TEXTLIST S2_Alarms
  0 = 'S2 0 Row 1 Failed To Advance.. Check Qxxx.x Default' | German: 'S2 0 Row 1 Failed To Advance.. Check Qxxx.x German' | French: 'S2 0 Row 1 Failed To Advance.. Check Qxxx.x French'
  1 = 'S2 1 Row 1 Failed To Return.. Check Qxxx.x Default' | German: 'S2 1 Row 1 Failed To Return.. Check Qxxx.x German' | French: 'S2 1 Row 1 Failed To Return.. Check Qxxx.x French'
  2 = 'S2 2 Row 1 Lost Advance Position... Check Ixxx.x Default' | German: 'S2 2 Row 1 Lost Advance Position... Check Ixxx.x German' | French: 'S2 2 Row 1 Lost Advance Position... Check Ixxx.x French'
  3 = 'S2 3 Row 1 Lost Return Position... Check Ixxx.x Default' | German: 'S2 3 Row 1 Lost Return Position... Check Ixxx.x German' | French: 'S2 3 Row 1 Lost Return Position... Check Ixxx.x French'
  4 = 'S2 4 Row 1 Switch Fault... Check Ixxx.x / Ixxx.x Default' | German: 'S2 4 Row 1 Switch Fault... Check Ixxx.x / Ixxx.x German' | French: 'S2 4 Row 1 Switch Fault... Check Ixxx.x / Ixxx.x French'
  5 = 'S2 5 Row 1 Spare Message Default' | German: 'S2 5 Row 1 Spare Message German' | French: 'S2 5 Row 1 Spare Message French'
  6 = 'S2 6 Row 1 Spare Message Default' | German: 'S2 6 Row 1 Spare Message German' | French: 'S2 6 Row 1 Spare Message French'
  7 = 'S2 7 Row 1 Spare Message Default' | German: 'S2 7 Row 1 Spare Message German' | French: 'S2 7 Row 1 Spare Message French'
  8 = 'S2 8 Row 1 Spare Message Default' | German: 'S2 8 Row 1 Spare Message German' | French: 'S2 8 Row 1 Spare Message French'
  9 = 'S2 9 Row 1 Spare Message Default' | German: 'S2 9 Row 1 Spare Message German' | French: 'S2 9 Row 1 Spare Message French'
  10 = 'S2 10 Row 2 Failed To Advance.. Check Qxxx.x Default' | German: 'S2 10 Row 2 Failed To Advance.. Check Qxxx.x German' | French: 'S2 10 Row 2 Failed To Advance.. Check Qxxx.x French'
  11 = 'S2 11 Row 2 Failed To Return.. Check Qxxx.x Default' | German: 'S2 11 Row 2 Failed To Return.. Check Qxxx.x German' | French: 'S2 11 Row 2 Failed To Return.. Check Qxxx.x French'
  12 = 'S2 12 Row 2 Lost Advance Position... Check Ixxx.x Default' | German: 'S2 12 Row 2 Lost Advance Position... Check Ixxx.x German' | French: 'S2 12 Row 2 Lost Advance Position... Check Ixxx.x French'
  13 = 'S2 13 Row 2 Lost Return Position... Check Ixxx.x Default' | German: 'S2 13 Row 2 Lost Return Position... Check Ixxx.x German' | French: 'S2 13 Row 2 Lost Return Position... Check Ixxx.x French'
  14 = 'S2 14 Row 2 Switch Fault... Check Ixxx.x / Ixxx.x Default' | German: 'S2 14 Row 2 Switch Fault... Check Ixxx.x / Ixxx.x German' | French: 'S2 14 Row 2 Switch Fault... Check Ixxx.x / Ixxx.x French'
  15 = 'S2 15 Row 2 Spare Message Default' | German: 'S2 15 Row 2 Spare Message German' | French: 'S2 15 Row 2 Spare Message French'
  16 = 'S2 16 Row 2 Spare Message Default' | German: 'S2 16 Row 2 Spare Message German' | French: 'S2 16 Row 2 Spare Message French'
  17 = 'S2 17 Row 2 Spare Message Default' | German: 'S2 17 Row 2 Spare Message German' | French: 'S2 17 Row 2 Spare Message French'
  18 = 'S2 18 Row 2 Spare Message Default' | German: 'S2 18 Row 2 Spare Message German' | French: 'S2 18 Row 2 Spare Message French'
  19 = 'S2 19 Row 2 Spare Message Default' | German: 'S2 19 Row 2 Spare Message German' | French: 'S2 19 Row 2 Spare Message French'
  20 = 'S2 20 Row 3 Failed To Advance.. Check Qxxx.x Default' | German: 'S2 20 Row 3 Failed To Advance.. Check Qxxx.x German' | French: 'S2 20 Row 3 Failed To Advance.. Check Qxxx.x French'
  21 = 'S2 21 Row 3 Failed To Return.. Check Qxxx.x Default' | German: 'S2 21 Row 3 Failed To Return.. Check Qxxx.x German' | French: 'S2 21 Row 3 Failed To Return.. Check Qxxx.x French'
  22 = 'S2 22 Row 3 Lost Advance Position... Check Ixxx.x Default' | German: 'S2 22 Row 3 Lost Advance Position... Check Ixxx.x German' | French: 'S2 22 Row 3 Lost Advance Position... Check Ixxx.x French'
  23 = 'S2 23 Row 3 Lost Return Position... Check Ixxx.x Default' | German: 'S2 23 Row 3 Lost Return Position... Check Ixxx.x German' | French: 'S2 23 Row 3 Lost Return Position... Check Ixxx.x French'
  24 = 'S2 24 Row 3 Switch Fault... Check Ixxx.x / Ixxx.x Default' | German: 'S2 24 Row 3 Switch Fault... Check Ixxx.x / Ixxx.x German' | French: 'S2 24 Row 3 Switch Fault... Check Ixxx.x / Ixxx.x French'
  25 = 'S2 25 Row 3 Spare Message Default' | German: 'S2 25 Row 3 Spare Message German' | French: 'S2 25 Row 3 Spare Message French'
  26 = 'S2 26 Row 3 Spare Message Default' | German: 'S2 26 Row 3 Spare Message German' | French: 'S2 26 Row 3 Spare Message French'
  27 = 'S2 27 Row 3 Spare Message Default' | German: 'S2 27 Row 3 Spare Message German' | French: 'S2 27 Row 3 Spare Message French'
  28 = 'S2 28 Row 3 Spare Message Default' | German: 'S2 28 Row 3 Spare Message German' | French: 'S2 28 Row 3 Spare Message French'
  29 = 'S2 29 Row 3 Spare Message Default' | German: 'S2 29 Row 3 Spare Message German' | French: 'S2 29 Row 3 Spare Message French'
  30 = 'S2 30 Row 4 Failed To Advance.. Check Qxxx.x Default' | German: 'S2 30 Row 4 Failed To Advance.. Check Qxxx.x German' | French: 'S2 30 Row 4 Failed To Advance.. Check Qxxx.x French'
  31 = 'S2 31 Row 4 Failed To Return.. Check Qxxx.x Default' | German: 'S2 31 Row 4 Failed To Return.. Check Qxxx.x German' | French: 'S2 31 Row 4 Failed To Return.. Check Qxxx.x French'
  32 = 'S2 32 Row 4 Lost Advance Position... Check Ixxx.x Default' | German: 'S2 32 Row 4 Lost Advance Position... Check Ixxx.x German' | French: 'S2 32 Row 4 Lost Advance Position... Check Ixxx.x French'
  33 = 'S2 33 Row 4 Lost Return Position... Check Ixxx.x Default' | German: 'S2 33 Row 4 Lost Return Position... Check Ixxx.x German' | French: 'S2 33 Row 4 Lost Return Position... Check Ixxx.x French'
  34 = 'S2 34 Row 4 Switch Fault... Check Ixxx.x / Ixxx.x Default' | German: 'S2 34 Row 4 Switch Fault... Check Ixxx.x / Ixxx.x German' | French: 'S2 34 Row 4 Switch Fault... Check Ixxx.x / Ixxx.x French'
  35 = 'S2 35 Row 4 Spare Message Default' | German: 'S2 35 Row 4 Spare Message German' | French: 'S2 35 Row 4 Spare Message French'
  36 = 'S2 36 Row 4 Spare Message Default' | German: 'S2 36 Row 4 Spare Message German' | French: 'S2 36 Row 4 Spare Message French'
  37 = 'S2 37 Row 4 Spare Message Default' | German: 'S2 37 Row 4 Spare Message German' | French: 'S2 37 Row 4 Spare Message French'
  38 = 'S2 38 Row 4 Spare Message Default' | German: 'S2 38 Row 4 Spare Message German' | French: 'S2 38 Row 4 Spare Message French'
  39 = 'S2 39 Row 4 Spare Message Default' | German: 'S2 39 Row 4 Spare Message German' | French: 'S2 39 Row 4 Spare Message French'
  40 = 'S2 40 Row 5 Failed To Advance.. Check Qxxx.x Default' | German: 'S2 40 Row 5 Failed To Advance.. Check Qxxx.x German' | French: 'S2 40 Row 5 Failed To Advance.. Check Qxxx.x French'
  41 = 'S2 41 Row 5 Failed To Return.. Check Qxxx.x Default' | German: 'S2 41 Row 5 Failed To Return.. Check Qxxx.x German' | French: 'S2 41 Row 5 Failed To Return.. Check Qxxx.x French'
  42 = 'S2 42 Row 5 Lost Advance Position... Check Ixxx.x Default' | German: 'S2 42 Row 5 Lost Advance Position... Check Ixxx.x German' | French: 'S2 42 Row 5 Lost Advance Position... Check Ixxx.x French'
  43 = 'S2 43 Row 5 Lost Return Position... Check Ixxx.x Default' | German: 'S2 43 Row 5 Lost Return Position... Check Ixxx.x German' | French: 'S2 43 Row 5 Lost Return Position... Check Ixxx.x French'
  44 = 'S2 44 Row 5 Switch Fault... Check Ixxx.x / Ixxx.x Default' | German: 'S2 44 Row 5 Switch Fault... Check Ixxx.x / Ixxx.x German' | French: 'S2 44 Row 5 Switch Fault... Check Ixxx.x / Ixxx.x French'
  45 = 'S2 45 Row 5 Spare Message Default' | German: 'S2 45 Row 5 Spare Message German' | French: 'S2 45 Row 5 Spare Message French'
  46 = 'S2 46 Row 5 Spare Message Default' | German: 'S2 46 Row 5 Spare Message German' | French: 'S2 46 Row 5 Spare Message French'
  47 = 'S2 47 Row 5 Spare Message Default' | German: 'S2 47 Row 5 Spare Message German' | French: 'S2 47 Row 5 Spare Message French'
  48 = 'S2 48 Row 5 Spare Message Default' | German: 'S2 48 Row 5 Spare Message German' | French: 'S2 48 Row 5 Spare Message French'
  49 = 'S2 49 Row 5 Spare Message Default' | German: 'S2 49 Row 5 Spare Message German' | French: 'S2 49 Row 5 Spare Message French'
  50 = 'S2 50 Row 6 Failed To Advance.. Check Qxxx.x Default' | German: 'S2 50 Row 6 Failed To Advance.. Check Qxxx.x German' | French: 'S2 50 Row 6 Failed To Advance.. Check Qxxx.x French'
  51 = 'S2 51 Row 6 Failed To Return.. Check Qxxx.x Default' | German: 'S2 51 Row 6 Failed To Return.. Check Qxxx.x German' | French: 'S2 51 Row 6 Failed To Return.. Check Qxxx.x French'
  52 = 'S2 52 Row 6 Lost Advance Position... Check Ixxx.x Default' | German: 'S2 52 Row 6 Lost Advance Position... Check Ixxx.x German' | French: 'S2 52 Row 6 Lost Advance Position... Check Ixxx.x French'
  53 = 'S2 53 Row 6 Lost Return Position... Check Ixxx.x Default' | German: 'S2 53 Row 6 Lost Return Position... Check Ixxx.x German' | French: 'S2 53 Row 6 Lost Return Position... Check Ixxx.x French'
  54 = 'S2 54 Row 6 Switch Fault... Check Ixxx.x / Ixxx.x Default' | German: 'S2 54 Row 6 Switch Fault... Check Ixxx.x / Ixxx.x German' | French: 'S2 54 Row 6 Switch Fault... Check Ixxx.x / Ixxx.x French'
  55 = 'S2 55 Row 6 Spare Message Default' | German: 'S2 55 Row 6 Spare Message German' | French: 'S2 55 Row 6 Spare Message French'
  56 = 'S2 56 Row 6 Spare Message Default' | German: 'S2 56 Row 6 Spare Message German' | French: 'S2 56 Row 6 Spare Message French'
  57 = 'S2 57 Row 6 Spare Message Default' | German: 'S2 57 Row 6 Spare Message German' | French: 'S2 57 Row 6 Spare Message French'
  58 = 'S2 58 Row 6 Spare Message Default' | German: 'S2 58 Row 6 Spare Message German' | French: 'S2 58 Row 6 Spare Message French'
  59 = 'S2 59 Row 6 Spare Message Default' | German: 'S2 59 Row 6 Spare Message German' | French: 'S2 59 Row 6 Spare Message French'
  60 = 'S2 60 Row 7 Failed To Advance.. Check Qxxx.x Default' | German: 'S2 60 Row 7 Failed To Advance.. Check Qxxx.x German' | French: 'S2 60 Row 7 Failed To Advance.. Check Qxxx.x French'
  61 = 'S2 61 Row 7 Failed To Return.. Check Qxxx.x Default' | German: 'S2 61 Row 7 Failed To Return.. Check Qxxx.x German' | French: 'S2 61 Row 7 Failed To Return.. Check Qxxx.x French'
  62 = 'S2 62 Row 7 Lost Advance Position... Check Ixxx.x Default' | German: 'S2 62 Row 7 Lost Advance Position... Check Ixxx.x German' | French: 'S2 62 Row 7 Lost Advance Position... Check Ixxx.x French'
  63 = 'S2 63 Row 7 Lost Return Position... Check Ixxx.x Default' | German: 'S2 63 Row 7 Lost Return Position... Check Ixxx.x German' | French: 'S2 63 Row 7 Lost Return Position... Check Ixxx.x French'
  64 = 'S2 64 Row 7 Switch Fault... Check Ixxx.x / Ixxx.x Default' | German: 'S2 64 Row 7 Switch Fault... Check Ixxx.x / Ixxx.x German' | French: 'S2 64 Row 7 Switch Fault... Check Ixxx.x / Ixxx.x French'
  65 = 'S2 65 Row 7 Spare Message Default' | German: 'S2 65 Row 7 Spare Message German' | French: 'S2 65 Row 7 Spare Message French'
  66 = 'S2 66 Row 7 Spare Message Default' | German: 'S2 66 Row 7 Spare Message German' | French: 'S2 66 Row 7 Spare Message French'
  67 = 'S2 67 Row 7 Spare Message Default' | German: 'S2 67 Row 7 Spare Message German' | French: 'S2 67 Row 7 Spare Message French'
  68 = 'S2 68 Row 7 Spare Message Default' | German: 'S2 68 Row 7 Spare Message German' | French: 'S2 68 Row 7 Spare Message French'
  69 = 'S2 69 Row 7 Spare Message Default' | German: 'S2 69 Row 7 Spare Message German' | French: 'S2 69 Row 7 Spare Message French'
  70 = 'S2 70 Row 8 Failed To Advance.. Check Qxxx.x Default' | German: 'S2 70 Row 8 Failed To Advance.. Check Qxxx.x German' | French: 'S2 70 Row 8 Failed To Advance.. Check Qxxx.x French'
  71 = 'S2 71 Row 8 Failed To Return.. Check Qxxx.x Default' | German: 'S2 71 Row 8 Failed To Return.. Check Qxxx.x German' | French: 'S2 71 Row 8 Failed To Return.. Check Qxxx.x French'
  72 = 'S2 72 Row 8 Lost Advance Position... Check Ixxx.x Default' | German: 'S2 72 Row 8 Lost Advance Position... Check Ixxx.x German' | French: 'S2 72 Row 8 Lost Advance Position... Check Ixxx.x French'
  73 = 'S2 73 Row 8 Lost Return Position... Check Ixxx.x Default' | German: 'S2 73 Row 8 Lost Return Position... Check Ixxx.x German' | French: 'S2 73 Row 8 Lost Return Position... Check Ixxx.x French'
  74 = 'S2 74 Row 8 Switch Fault... Check Ixxx.x / Ixxx.x Default' | German: 'S2 74 Row 8 Switch Fault... Check Ixxx.x / Ixxx.x German' | French: 'S2 74 Row 8 Switch Fault... Check Ixxx.x / Ixxx.x French'
  75 = 'S2 75 Row 8 Spare Message Default' | German: 'S2 75 Row 8 Spare Message German' | French: 'S2 75 Row 8 Spare Message French'
  76 = 'S2 76 Row 8 Spare Message Default' | German: 'S2 76 Row 8 Spare Message German' | French: 'S2 76 Row 8 Spare Message French'
  77 = 'S2 77 Row 8 Spare Message Default' | German: 'S2 77 Row 8 Spare Message German' | French: 'S2 77 Row 8 Spare Message French'
  78 = 'S2 78 Row 8 Spare Message Default' | German: 'S2 78 Row 8 Spare Message German' | French: 'S2 78 Row 8 Spare Message French'
  79 = 'S2 79 Row 8 Spare Message Default' | German: 'S2 79 Row 8 Spare Message German' | French: 'S2 79 Row 8 Spare Message French'
  80 = 'S2 80 Row 9 Failed To Advance.. Check Qxxx.x Default' | German: 'S2 80 Row 9 Failed To Advance.. Check Qxxx.x German' | French: 'S2 80 Row 9 Failed To Advance.. Check Qxxx.x French'
  81 = 'S2 81 Row 9 Failed To Return.. Check Qxxx.x Default' | German: 'S2 81 Row 9 Failed To Return.. Check Qxxx.x German' | French: 'S2 81 Row 9 Failed To Return.. Check Qxxx.x French'
  82 = 'S2 82 Row 9 Lost Advance Position... Check Ixxx.x Default' | German: 'S2 82 Row 9 Lost Advance Position... Check Ixxx.x German' | French: 'S2 82 Row 9 Lost Advance Position... Check Ixxx.x French'
  83 = 'S2 83 Row 9 Lost Return Position... Check Ixxx.x Default' | German: 'S2 83 Row 9 Lost Return Position... Check Ixxx.x German' | French: 'S2 83 Row 9 Lost Return Position... Check Ixxx.x French'
  84 = 'S2 84 Row 9 Switch Fault... Check Ixxx.x / Ixxx.x Default' | German: 'S2 84 Row 9 Switch Fault... Check Ixxx.x / Ixxx.x German' | French: 'S2 84 Row 9 Switch Fault... Check Ixxx.x / Ixxx.x French'
  85 = 'S2 85 Row 9 Spare Message Default' | German: 'S2 85 Row 9 Spare Message German' | French: 'S2 85 Row 9 Spare Message French'
  86 = 'S2 86 Row 9 Spare Message Default' | German: 'S2 86 Row 9 Spare Message German' | French: 'S2 86 Row 9 Spare Message French'
  87 = 'S2 87 Row 9 Spare Message Default' | German: 'S2 87 Row 9 Spare Message German' | French: 'S2 87 Row 9 Spare Message French'
  88 = 'S2 88 Row 9 Spare Message Default' | German: 'S2 88 Row 9 Spare Message German' | French: 'S2 88 Row 9 Spare Message French'
  89 = 'S2 89 Row 9 Spare Message Default' | German: 'S2 89 Row 9 Spare Message German' | French: 'S2 89 Row 9 Spare Message French'
  90 = 'S2 90 Row 10 Failed To Advance.. Check Qxxx.x Default' | German: 'S2 90 Row 10 Failed To Advance.. Check Qxxx.x German' | French: 'S2 90 Row 10 Failed To Advance.. Check Qxxx.x French'
  91 = 'S2 91 Row 10 Failed To Return.. Check Qxxx.x Default' | German: 'S2 91 Row 10 Failed To Return.. Check Qxxx.x German' | French: 'S2 91 Row 10 Failed To Return.. Check Qxxx.x French'
  92 = 'S2 92 Row 10 Lost Advance Position... Check Ixxx.x Default' | German: 'S2 92 Row 10 Lost Advance Position... Check Ixxx.x German' | French: 'S2 92 Row 10 Lost Advance Position... Check Ixxx.x French'
  93 = 'S2 93 Row 10 Lost Return Position... Check Ixxx.x Default' | German: 'S2 93 Row 10 Lost Return Position... Check Ixxx.x German' | French: 'S2 93 Row 10 Lost Return Position... Check Ixxx.x French'
  94 = 'S2 94 Row 10 Switch Fault... Check Ixxx.x / Ixxx.x Default' | German: 'S2 94 Row 10 Switch Fault... Check Ixxx.x / Ixxx.x German' | French: 'S2 94 Row 10 Switch Fault... Check Ixxx.x / Ixxx.x French'
  95 = 'S2 95 Row 10 Spare Message Default' | German: 'S2 95 Row 10 Spare Message German' | French: 'S2 95 Row 10 Spare Message French'
  96 = 'S2 96 Row 10 Spare Message Default' | German: 'S2 96 Row 10 Spare Message German' | French: 'S2 96 Row 10 Spare Message French'
  97 = 'S2 97 Row 10 Spare Message Default' | German: 'S2 97 Row 10 Spare Message German' | French: 'S2 97 Row 10 Spare Message French'
  98 = 'S2 98 Row 10 Spare Message Default' | German: 'S2 98 Row 10 Spare Message German' | French: 'S2 98 Row 10 Spare Message French'
  99 = 'S2 99 Row 10 Spare Message Default' | German: 'S2 99 Row 10 Spare Message German' | French: 'S2 99 Row 10 Spare Message French'
  100 = 'S2 100 Row 11 Failed To Advance.. Check Qxxx.x Default' | German: 'S2 100 Row 11 Failed To Advance.. Check Qxxx.x German' | French: 'S2 100 Row 11 Failed To Advance.. Check Qxxx.x French'
  101 = 'S2 101 Row 11 Failed To Return.. Check Qxxx.x Default' | German: 'S2 101 Row 11 Failed To Return.. Check Qxxx.x German' | French: 'S2 101 Row 11 Failed To Return.. Check Qxxx.x French'
  102 = 'S2 102 Row 11 Lost Advance Position... Check Ixxx.x Default' | German: 'S2 102 Row 11 Lost Advance Position... Check Ixxx.x German' | French: 'S2 102 Row 11 Lost Advance Position... Check Ixxx.x French'
  103 = 'S2 103 Row 11 Lost Return Position... Check Ixxx.x Default' | German: 'S2 103 Row 11 Lost Return Position... Check Ixxx.x German' | French: 'S2 103 Row 11 Lost Return Position... Check Ixxx.x French'
  104 = 'S2 104 Row 11 Switch Fault... Check Ixxx.x / Ixxx.x Default' | German: 'S2 104 Row 11 Switch Fault... Check Ixxx.x / Ixxx.x German' | French: 'S2 104 Row 11 Switch Fault... Check Ixxx.x / Ixxx.x French'
  105 = 'S2 105 Row 11 Spare Message Default' | German: 'S2 105 Row 11 Spare Message German' | French: 'S2 105 Row 11 Spare Message French'
  106 = 'S2 106 Row 11 Spare Message Default' | German: 'S2 106 Row 11 Spare Message German' | French: 'S2 106 Row 11 Spare Message French'
  107 = 'S2 107 Row 11 Spare Message Default' | German: 'S2 107 Row 11 Spare Message German' | French: 'S2 107 Row 11 Spare Message French'
  108 = 'S2 108 Row 11 Spare Message Default' | German: 'S2 108 Row 11 Spare Message German' | French: 'S2 108 Row 11 Spare Message French'
  109 = 'S2 109 Row 11 Spare Message Default' | German: 'S2 109 Row 11 Spare Message German' | French: 'S2 109 Row 11 Spare Message French'
  110 = 'S2 110 Row 12 Failed To Advance.. Check Qxxx.x Default' | German: 'S2 110 Row 12 Failed To Advance.. Check Qxxx.x German' | French: 'S2 110 Row 12 Failed To Advance.. Check Qxxx.x French'
  111 = 'S2 111 Row 12 Failed To Return.. Check Qxxx.x Default' | German: 'S2 111 Row 12 Failed To Return.. Check Qxxx.x German' | French: 'S2 111 Row 12 Failed To Return.. Check Qxxx.x French'
  112 = 'S2 112 Row 12 Lost Advance Position... Check Ixxx.x Default' | German: 'S2 112 Row 12 Lost Advance Position... Check Ixxx.x German' | French: 'S2 112 Row 12 Lost Advance Position... Check Ixxx.x French'
  113 = 'S2 113 Row 12 Lost Return Position... Check Ixxx.x Default' | German: 'S2 113 Row 12 Lost Return Position... Check Ixxx.x German' | French: 'S2 113 Row 12 Lost Return Position... Check Ixxx.x French'
  114 = 'S2 114 Row 12 Switch Fault... Check Ixxx.x / Ixxx.x Default' | German: 'S2 114 Row 12 Switch Fault... Check Ixxx.x / Ixxx.x German' | French: 'S2 114 Row 12 Switch Fault... Check Ixxx.x / Ixxx.x French'
  115 = 'S2 115 Row 12 Spare Message Default' | German: 'S2 115 Row 12 Spare Message German' | French: 'S2 115 Row 12 Spare Message French'
  116 = 'S2 116 Row 12 Spare Message Default' | German: 'S2 116 Row 12 Spare Message German' | French: 'S2 116 Row 12 Spare Message French'
  117 = 'S2 117 Row 12 Spare Message Default' | German: 'S2 117 Row 12 Spare Message German' | French: 'S2 117 Row 12 Spare Message French'
  118 = 'S2 118 Row 12 Spare Message Default' | German: 'S2 118 Row 12 Spare Message German' | French: 'S2 118 Row 12 Spare Message French'
  119 = 'S2 119 Row 12 Spare Message Default' | German: 'S2 119 Row 12 Spare Message German' | French: 'S2 119 Row 12 Spare Message French'
  120 = 'S2 120 Row 13 Failed To Advance.. Check Qxxx.x Default' | German: 'S2 120 Row 13 Failed To Advance.. Check Qxxx.x German' | French: 'S2 120 Row 13 Failed To Advance.. Check Qxxx.x French'
  121 = 'S2 121 Row 13 Failed To Return.. Check Qxxx.x Default' | German: 'S2 121 Row 13 Failed To Return.. Check Qxxx.x German' | French: 'S2 121 Row 13 Failed To Return.. Check Qxxx.x French'
  122 = 'S2 122 Row 13 Lost Advance Position... Check Ixxx.x Default' | German: 'S2 122 Row 13 Lost Advance Position... Check Ixxx.x German' | French: 'S2 122 Row 13 Lost Advance Position... Check Ixxx.x French'
  123 = 'S2 123 Row 13 Lost Return Position... Check Ixxx.x Default' | German: 'S2 123 Row 13 Lost Return Position... Check Ixxx.x German' | French: 'S2 123 Row 13 Lost Return Position... Check Ixxx.x French'
  124 = 'S2 124 Row 13 Switch Fault... Check Ixxx.x / Ixxx.x Default' | German: 'S2 124 Row 13 Switch Fault... Check Ixxx.x / Ixxx.x German' | French: 'S2 124 Row 13 Switch Fault... Check Ixxx.x / Ixxx.x French'
  125 = 'S2 125 Row 13 Spare Message Default' | German: 'S2 125 Row 13 Spare Message German' | French: 'S2 125 Row 13 Spare Message French'
  126 = 'S2 126 Row 13 Spare Message Default' | German: 'S2 126 Row 13 Spare Message German' | French: 'S2 126 Row 13 Spare Message French'
  127 = 'S2 127 Row 13 Spare Message Default' | German: 'S2 127 Row 13 Spare Message German' | French: 'S2 127 Row 13 Spare Message French'
  128 = 'S2 128 Row 13 Spare Message Default' | German: 'S2 128 Row 13 Spare Message German' | French: 'S2 128 Row 13 Spare Message French'
  129 = 'S2 129 Row 13 Spare Message Default' | German: 'S2 129 Row 13 Spare Message German' | French: 'S2 129 Row 13 Spare Message French'
  130 = 'S2 130 Row 14 Failed To Advance.. Check Qxxx.x Default' | German: 'S2 130 Row 14 Failed To Advance.. Check Qxxx.x German' | French: 'S2 130 Row 14 Failed To Advance.. Check Qxxx.x French'
  131 = 'S2 131 Row 14 Failed To Return.. Check Qxxx.x Default' | German: 'S2 131 Row 14 Failed To Return.. Check Qxxx.x German' | French: 'S2 131 Row 14 Failed To Return.. Check Qxxx.x French'
  132 = 'S2 132 Row 14 Lost Advance Position... Check Ixxx.x Default' | German: 'S2 132 Row 14 Lost Advance Position... Check Ixxx.x German' | French: 'S2 132 Row 14 Lost Advance Position... Check Ixxx.x French'
  133 = 'S2 133 Row 14 Lost Return Position... Check Ixxx.x Default' | German: 'S2 133 Row 14 Lost Return Position... Check Ixxx.x German' | French: 'S2 133 Row 14 Lost Return Position... Check Ixxx.x French'
  134 = 'S2 134 Row 14 Switch Fault... Check Ixxx.x / Ixxx.x Default' | German: 'S2 134 Row 14 Switch Fault... Check Ixxx.x / Ixxx.x German' | French: 'S2 134 Row 14 Switch Fault... Check Ixxx.x / Ixxx.x French'
  135 = 'S2 135 Row 14 Spare Message Default' | German: 'S2 135 Row 14 Spare Message German' | French: 'S2 135 Row 14 Spare Message French'
  136 = 'S2 136 Row 14 Spare Message Default' | German: 'S2 136 Row 14 Spare Message German' | French: 'S2 136 Row 14 Spare Message French'
  137 = 'S2 137 Row 14 Spare Message Default' | German: 'S2 137 Row 14 Spare Message German' | French: 'S2 137 Row 14 Spare Message French'
  138 = 'S2 138 Row 14 Spare Message Default' | German: 'S2 138 Row 14 Spare Message German' | French: 'S2 138 Row 14 Spare Message French'
  139 = 'S2 139 Row 14 Spare Message Default' | German: 'S2 139 Row 14 Spare Message German' | French: 'S2 139 Row 14 Spare Message French'
  140 = 'S2 140 Row 15 Failed To Advance.. Check Qxxx.x Default' | German: 'S2 140 Row 15 Failed To Advance.. Check Qxxx.x German' | French: 'S2 140 Row 15 Failed To Advance.. Check Qxxx.x French'
  141 = 'S2 141 Row 15 Failed To Return.. Check Qxxx.x Default' | German: 'S2 141 Row 15 Failed To Return.. Check Qxxx.x German' | French: 'S2 141 Row 15 Failed To Return.. Check Qxxx.x French'
  142 = 'S2 142 Row 15 Lost Advance Position... Check Ixxx.x Default' | German: 'S2 142 Row 15 Lost Advance Position... Check Ixxx.x German' | French: 'S2 142 Row 15 Lost Advance Position... Check Ixxx.x French'
  143 = 'S2 143 Row 15 Lost Return Position... Check Ixxx.x Default' | German: 'S2 143 Row 15 Lost Return Position... Check Ixxx.x German' | French: 'S2 143 Row 15 Lost Return Position... Check Ixxx.x French'
  144 = 'S2 144 Row 15 Switch Fault... Check Ixxx.x / Ixxx.x Default' | German: 'S2 144 Row 15 Switch Fault... Check Ixxx.x / Ixxx.x German' | French: 'S2 144 Row 15 Switch Fault... Check Ixxx.x / Ixxx.x French'
  145 = 'S2 145 Row 15 Spare Message Default' | German: 'S2 145 Row 15 Spare Message German' | French: 'S2 145 Row 15 Spare Message French'
  146 = 'S2 146 Row 15 Spare Message Default' | German: 'S2 146 Row 15 Spare Message German' | French: 'S2 146 Row 15 Spare Message French'
  147 = 'S2 147 Row 15 Spare Message Default' | German: 'S2 147 Row 15 Spare Message German' | French: 'S2 147 Row 15 Spare Message French'
  148 = 'S2 148 Row 15 Spare Message Default' | German: 'S2 148 Row 15 Spare Message German' | French: 'S2 148 Row 15 Spare Message French'
  149 = 'S2 149 Row 15 Spare Message Default' | German: 'S2 149 Row 15 Spare Message German' | French: 'S2 149 Row 15 Spare Message French'
  150 = 'S2 150 Row 16 Failed To Advance.. Check Qxxx.x Default' | German: 'S2 150 Row 16 Failed To Advance.. Check Qxxx.x German' | French: 'S2 150 Row 16 Failed To Advance.. Check Qxxx.x French'
  151 = 'S2 151 Row 16 Failed To Return.. Check Qxxx.x Default' | German: 'S2 151 Row 16 Failed To Return.. Check Qxxx.x German' | French: 'S2 151 Row 16 Failed To Return.. Check Qxxx.x French'
  152 = 'S2 152 Row 16 Lost Advance Position... Check Ixxx.x Default' | German: 'S2 152 Row 16 Lost Advance Position... Check Ixxx.x German' | French: 'S2 152 Row 16 Lost Advance Position... Check Ixxx.x French'
  153 = 'S2 153 Row 16 Lost Return Position... Check Ixxx.x Default' | German: 'S2 153 Row 16 Lost Return Position... Check Ixxx.x German' | French: 'S2 153 Row 16 Lost Return Position... Check Ixxx.x French'
  154 = 'S2 154 Row 16 Switch Fault... Check Ixxx.x / Ixxx.x Default' | German: 'S2 154 Row 16 Switch Fault... Check Ixxx.x / Ixxx.x German' | French: 'S2 154 Row 16 Switch Fault... Check Ixxx.x / Ixxx.x French'
  155 = 'S2 155 Row 16 Spare Message Default' | German: 'S2 155 Row 16 Spare Message German' | French: 'S2 155 Row 16 Spare Message French'
  156 = 'S2 156 Row 16 Spare Message Default' | German: 'S2 156 Row 16 Spare Message German' | French: 'S2 156 Row 16 Spare Message French'
  157 = 'S2 157 Row 16 Spare Message Default' | German: 'S2 157 Row 16 Spare Message German' | French: 'S2 157 Row 16 Spare Message French'
  158 = 'S2 158 Row 16 Spare Message Default' | German: 'S2 158 Row 16 Spare Message German' | French: 'S2 158 Row 16 Spare Message French'
  159 = 'S2 159 Row 16 Spare Message Default' | German: 'S2 159 Row 16 Spare Message German' | French: 'S2 159 Row 16 Spare Message French'
  160 = 'S2 160 Row 17 Failed To Advance.. Check Qxxx.x Default' | German: 'S2 160 Row 17 Failed To Advance.. Check Qxxx.x German' | French: 'S2 160 Row 17 Failed To Advance.. Check Qxxx.x French'
  161 = 'S2 161 Row 17 Failed To Return.. Check Qxxx.x Default' | German: 'S2 161 Row 17 Failed To Return.. Check Qxxx.x German' | French: 'S2 161 Row 17 Failed To Return.. Check Qxxx.x French'
  162 = 'S2 162 Row 17 Lost Advance Position... Check Ixxx.x Default' | German: 'S2 162 Row 17 Lost Advance Position... Check Ixxx.x German' | French: 'S2 162 Row 17 Lost Advance Position... Check Ixxx.x French'
  163 = 'S2 163 Row 17 Lost Return Position... Check Ixxx.x Default' | German: 'S2 163 Row 17 Lost Return Position... Check Ixxx.x German' | French: 'S2 163 Row 17 Lost Return Position... Check Ixxx.x French'
  164 = 'S2 164 Row 17 Switch Fault... Check Ixxx.x / Ixxx.x Default' | German: 'S2 164 Row 17 Switch Fault... Check Ixxx.x / Ixxx.x German' | French: 'S2 164 Row 17 Switch Fault... Check Ixxx.x / Ixxx.x French'
  165 = 'S2 165 Row 17 Spare Message Default' | German: 'S2 165 Row 17 Spare Message German' | French: 'S2 165 Row 17 Spare Message French'
  166 = 'S2 166 Row 17 Spare Message Default' | German: 'S2 166 Row 17 Spare Message German' | French: 'S2 166 Row 17 Spare Message French'
  167 = 'S2 167 Row 17 Spare Message Default' | German: 'S2 167 Row 17 Spare Message German' | French: 'S2 167 Row 17 Spare Message French'
  168 = 'S2 168 Row 17 Spare Message Default' | German: 'S2 168 Row 17 Spare Message German' | French: 'S2 168 Row 17 Spare Message French'
  169 = 'S2 169 Row 17 Spare Message Default' | German: 'S2 169 Row 17 Spare Message German' | French: 'S2 169 Row 17 Spare Message French'
  170 = 'S2 170 Row 18 Failed To Advance.. Check Qxxx.x Default' | German: 'S2 170 Row 18 Failed To Advance.. Check Qxxx.x German' | French: 'S2 170 Row 18 Failed To Advance.. Check Qxxx.x French'
  171 = 'S2 171 Row 18 Failed To Return.. Check Qxxx.x Default' | German: 'S2 171 Row 18 Failed To Return.. Check Qxxx.x German' | French: 'S2 171 Row 18 Failed To Return.. Check Qxxx.x French'
  172 = 'S2 172 Row 18 Lost Advance Position... Check Ixxx.x Default' | German: 'S2 172 Row 18 Lost Advance Position... Check Ixxx.x German' | French: 'S2 172 Row 18 Lost Advance Position... Check Ixxx.x French'
  173 = 'S2 173 Row 18 Lost Return Position... Check Ixxx.x Default' | German: 'S2 173 Row 18 Lost Return Position... Check Ixxx.x German' | French: 'S2 173 Row 18 Lost Return Position... Check Ixxx.x French'
  174 = 'S2 174 Row 18 Switch Fault... Check Ixxx.x / Ixxx.x Default' | German: 'S2 174 Row 18 Switch Fault... Check Ixxx.x / Ixxx.x German' | French: 'S2 174 Row 18 Switch Fault... Check Ixxx.x / Ixxx.x French'
  175 = 'S2 175 Row 18 Spare Message Default' | German: 'S2 175 Row 18 Spare Message German' | French: 'S2 175 Row 18 Spare Message French'
  176 = 'S2 176 Row 18 Spare Message Default' | German: 'S2 176 Row 18 Spare Message German' | French: 'S2 176 Row 18 Spare Message French'
  177 = 'S2 177 Row 18 Spare Message Default' | German: 'S2 177 Row 18 Spare Message German' | French: 'S2 177 Row 18 Spare Message French'
  178 = 'S2 178 Row 18 Spare Message Default' | German: 'S2 178 Row 18 Spare Message German' | French: 'S2 178 Row 18 Spare Message French'
  179 = 'S2 179 Row 18 Spare Message Default' | German: 'S2 179 Row 18 Spare Message German' | French: 'S2 179 Row 18 Spare Message French'
  180 = 'S2 180 Row 19 Failed To Advance.. Check Qxxx.x Default' | German: 'S2 180 Row 19 Failed To Advance.. Check Qxxx.x German' | French: 'S2 180 Row 19 Failed To Advance.. Check Qxxx.x French'
  181 = 'S2 181 Row 19 Failed To Return.. Check Qxxx.x Default' | German: 'S2 181 Row 19 Failed To Return.. Check Qxxx.x German' | French: 'S2 181 Row 19 Failed To Return.. Check Qxxx.x French'
  182 = 'S2 182 Row 19 Lost Advance Position... Check Ixxx.x Default' | German: 'S2 182 Row 19 Lost Advance Position... Check Ixxx.x German' | French: 'S2 182 Row 19 Lost Advance Position... Check Ixxx.x French'
  183 = 'S2 183 Row 19 Lost Return Position... Check Ixxx.x Default' | German: 'S2 183 Row 19 Lost Return Position... Check Ixxx.x German' | French: 'S2 183 Row 19 Lost Return Position... Check Ixxx.x French'
  184 = 'S2 184 Row 19 Switch Fault... Check Ixxx.x / Ixxx.x Default' | German: 'S2 184 Row 19 Switch Fault... Check Ixxx.x / Ixxx.x German' | French: 'S2 184 Row 19 Switch Fault... Check Ixxx.x / Ixxx.x French'
  185 = 'S2 185 Row 19 Spare Message Default' | German: 'S2 185 Row 19 Spare Message German' | French: 'S2 185 Row 19 Spare Message French'
  186 = 'S2 186 Row 19 Spare Message Default' | German: 'S2 186 Row 19 Spare Message German' | French: 'S2 186 Row 19 Spare Message French'
  187 = 'S2 187 Row 19 Spare Message Default' | German: 'S2 187 Row 19 Spare Message German' | French: 'S2 187 Row 19 Spare Message French'
  188 = 'S2 188 Row 19 Spare Message Default' | German: 'S2 188 Row 19 Spare Message German' | French: 'S2 188 Row 19 Spare Message French'
  189 = 'S2 189 Row 19 Spare Message Default' | German: 'S2 189 Row 19 Spare Message German' | French: 'S2 189 Row 19 Spare Message French'
  190 = 'S2 190 Row 20 Failed To Advance.. Check Qxxx.x Default' | German: 'S2 190 Row 20 Failed To Advance.. Check Qxxx.x German' | French: 'S2 190 Row 20 Failed To Advance.. Check Qxxx.x French'
  191 = 'S2 191 Row 20 Failed To Return.. Check Qxxx.x Default' | German: 'S2 191 Row 20 Failed To Return.. Check Qxxx.x German' | French: 'S2 191 Row 20 Failed To Return.. Check Qxxx.x French'
  192 = 'S2 192 Row 20 Lost Advance Position... Check Ixxx.x Default' | German: 'S2 192 Row 20 Lost Advance Position... Check Ixxx.x German' | French: 'S2 192 Row 20 Lost Advance Position... Check Ixxx.x French'
  193 = 'S2 193 Row 20 Lost Return Position... Check Ixxx.x Default' | German: 'S2 193 Row 20 Lost Return Position... Check Ixxx.x German' | French: 'S2 193 Row 20 Lost Return Position... Check Ixxx.x French'
  194 = 'S2 194 Row 20 Switch Fault... Check Ixxx.x / Ixxx.x Default' | German: 'S2 194 Row 20 Switch Fault... Check Ixxx.x / Ixxx.x German' | French: 'S2 194 Row 20 Switch Fault... Check Ixxx.x / Ixxx.x French'
  195 = 'S2 195 Row 20 Spare Message Default' | German: 'S2 195 Row 20 Spare Message German' | French: 'S2 195 Row 20 Spare Message French'
  196 = 'S2 196 Row 20 Spare Message Default' | German: 'S2 196 Row 20 Spare Message German' | French: 'S2 196 Row 20 Spare Message French'
  197 = 'S2 197 Row 20 Spare Message Default' | German: 'S2 197 Row 20 Spare Message German' | French: 'S2 197 Row 20 Spare Message French'
  198 = 'S2 198 Row 20 Spare Message Default' | German: 'S2 198 Row 20 Spare Message German' | French: 'S2 198 Row 20 Spare Message French'
  199 = 'S2 199 Row 20 Spare Message Default' | German: 'S2 199 Row 20 Spare Message German' | French: 'S2 199 Row 20 Spare Message French'
  200 = 'S2 200 Row 21 Failed To Advance.. Check Qxxx.x Default' | German: 'S2 200 Row 21 Failed To Advance.. Check Qxxx.x German' | French: 'S2 200 Row 21 Failed To Advance.. Check Qxxx.x French'
  201 = 'S2 201 Row 21 Failed To Return.. Check Qxxx.x Default' | German: 'S2 201 Row 21 Failed To Return.. Check Qxxx.x German' | French: 'S2 201 Row 21 Failed To Return.. Check Qxxx.x French'
  202 = 'S2 202 Row 21 Lost Advance Position... Check Ixxx.x Default' | German: 'S2 202 Row 21 Lost Advance Position... Check Ixxx.x German' | French: 'S2 202 Row 21 Lost Advance Position... Check Ixxx.x French'
  203 = 'S2 203 Row 21 Lost Return Position... Check Ixxx.x Default' | German: 'S2 203 Row 21 Lost Return Position... Check Ixxx.x German' | French: 'S2 203 Row 21 Lost Return Position... Check Ixxx.x French'
  204 = 'S2 204 Row 21 Switch Fault... Check Ixxx.x / Ixxx.x Default' | German: 'S2 204 Row 21 Switch Fault... Check Ixxx.x / Ixxx.x German' | French: 'S2 204 Row 21 Switch Fault... Check Ixxx.x / Ixxx.x French'
  205 = 'S2 205 Row 21 Spare Message Default' | German: 'S2 205 Row 21 Spare Message German' | French: 'S2 205 Row 21 Spare Message French'
  206 = 'S2 206 Row 21 Spare Message Default' | German: 'S2 206 Row 21 Spare Message German' | French: 'S2 206 Row 21 Spare Message French'
  207 = 'S2 207 Row 21 Spare Message Default' | German: 'S2 207 Row 21 Spare Message German' | French: 'S2 207 Row 21 Spare Message French'
  208 = 'S2 208 Row 21 Spare Message Default' | German: 'S2 208 Row 21 Spare Message German' | French: 'S2 208 Row 21 Spare Message French'
  209 = 'S2 209 Row 21 Spare Message Default' | German: 'S2 209 Row 21 Spare Message German' | French: 'S2 209 Row 21 Spare Message French'
  210 = 'S2 210 Row 22 Failed To Advance.. Check Qxxx.x Default' | German: 'S2 210 Row 22 Failed To Advance.. Check Qxxx.x German' | French: 'S2 210 Row 22 Failed To Advance.. Check Qxxx.x French'
  211 = 'S2 211 Row 22 Failed To Return.. Check Qxxx.x Default' | German: 'S2 211 Row 22 Failed To Return.. Check Qxxx.x German' | French: 'S2 211 Row 22 Failed To Return.. Check Qxxx.x French'
  212 = 'S2 212 Row 22 Lost Advance Position... Check Ixxx.x Default' | German: 'S2 212 Row 22 Lost Advance Position... Check Ixxx.x German' | French: 'S2 212 Row 22 Lost Advance Position... Check Ixxx.x French'
  213 = 'S2 213 Row 22 Lost Return Position... Check Ixxx.x Default' | German: 'S2 213 Row 22 Lost Return Position... Check Ixxx.x German' | French: 'S2 213 Row 22 Lost Return Position... Check Ixxx.x French'
  214 = 'S2 214 Row 22 Switch Fault... Check Ixxx.x / Ixxx.x Default' | German: 'S2 214 Row 22 Switch Fault... Check Ixxx.x / Ixxx.x German' | French: 'S2 214 Row 22 Switch Fault... Check Ixxx.x / Ixxx.x French'
  215 = 'S2 215 Row 22 Spare Message Default' | German: 'S2 215 Row 22 Spare Message German' | French: 'S2 215 Row 22 Spare Message French'
  216 = 'S2 216 Row 22 Spare Message Default' | German: 'S2 216 Row 22 Spare Message German' | French: 'S2 216 Row 22 Spare Message French'
  217 = 'S2 217 Row 22 Spare Message Default' | German: 'S2 217 Row 22 Spare Message German' | French: 'S2 217 Row 22 Spare Message French'
  218 = 'S2 218 Row 22 Spare Message Default' | German: 'S2 218 Row 22 Spare Message German' | French: 'S2 218 Row 22 Spare Message French'
  219 = 'S2 219 Row 22 Spare Message Default' | German: 'S2 219 Row 22 Spare Message German' | French: 'S2 219 Row 22 Spare Message French'
  220 = 'S2 220 Row 23 Failed To Advance.. Check Qxxx.x Default' | German: 'S2 220 Row 23 Failed To Advance.. Check Qxxx.x German' | French: 'S2 220 Row 23 Failed To Advance.. Check Qxxx.x French'
  221 = 'S2 221 Row 23 Failed To Return.. Check Qxxx.x Default' | German: 'S2 221 Row 23 Failed To Return.. Check Qxxx.x German' | French: 'S2 221 Row 23 Failed To Return.. Check Qxxx.x French'
  222 = 'S2 222 Row 23 Lost Advance Position... Check Ixxx.x Default' | German: 'S2 222 Row 23 Lost Advance Position... Check Ixxx.x German' | French: 'S2 222 Row 23 Lost Advance Position... Check Ixxx.x French'
  223 = 'S2 223 Row 23 Lost Return Position... Check Ixxx.x Default' | German: 'S2 223 Row 23 Lost Return Position... Check Ixxx.x German' | French: 'S2 223 Row 23 Lost Return Position... Check Ixxx.x French'
  224 = 'S2 224 Row 23 Switch Fault... Check Ixxx.x / Ixxx.x Default' | German: 'S2 224 Row 23 Switch Fault... Check Ixxx.x / Ixxx.x German' | French: 'S2 224 Row 23 Switch Fault... Check Ixxx.x / Ixxx.x French'
  225 = 'S2 225 Row 23 Spare Message Default' | German: 'S2 225 Row 23 Spare Message German' | French: 'S2 225 Row 23 Spare Message French'
  226 = 'S2 226 Row 23 Spare Message Default' | German: 'S2 226 Row 23 Spare Message German' | French: 'S2 226 Row 23 Spare Message French'
  227 = 'S2 227 Row 23 Spare Message Default' | German: 'S2 227 Row 23 Spare Message German' | French: 'S2 227 Row 23 Spare Message French'
  228 = 'S2 228 Row 23 Spare Message Default' | German: 'S2 228 Row 23 Spare Message German' | French: 'S2 228 Row 23 Spare Message French'
  229 = 'S2 229 Row 23 Spare Message Default' | German: 'S2 229 Row 23 Spare Message German' | French: 'S2 229 Row 23 Spare Message French'
  230 = 'S2 230 Row 24 Failed To Advance.. Check Qxxx.x Default' | German: 'S2 230 Row 24 Failed To Advance.. Check Qxxx.x German' | French: 'S2 230 Row 24 Failed To Advance.. Check Qxxx.x French'
  231 = 'S2 231 Row 24 Failed To Return.. Check Qxxx.x Default' | German: 'S2 231 Row 24 Failed To Return.. Check Qxxx.x German' | French: 'S2 231 Row 24 Failed To Return.. Check Qxxx.x French'
  232 = 'S2 232 Row 24 Lost Advance Position... Check Ixxx.x Default' | German: 'S2 232 Row 24 Lost Advance Position... Check Ixxx.x German' | French: 'S2 232 Row 24 Lost Advance Position... Check Ixxx.x French'
  233 = 'S2 233 Row 24 Lost Return Position... Check Ixxx.x Default' | German: 'S2 233 Row 24 Lost Return Position... Check Ixxx.x German' | French: 'S2 233 Row 24 Lost Return Position... Check Ixxx.x French'
  234 = 'S2 234 Row 24 Switch Fault... Check Ixxx.x / Ixxx.x Default' | German: 'S2 234 Row 24 Switch Fault... Check Ixxx.x / Ixxx.x German' | French: 'S2 234 Row 24 Switch Fault... Check Ixxx.x / Ixxx.x French'
  235 = 'S2 235 Row 24 Spare Message Default' | German: 'S2 235 Row 24 Spare Message German' | French: 'S2 235 Row 24 Spare Message French'
  236 = 'S2 236 Row 24 Spare Message Default' | German: 'S2 236 Row 24 Spare Message German' | French: 'S2 236 Row 24 Spare Message French'
  237 = 'S2 237 Row 24 Spare Message Default' | German: 'S2 237 Row 24 Spare Message German' | French: 'S2 237 Row 24 Spare Message French'
  238 = 'S2 238 Row 24 Spare Message Default' | German: 'S2 238 Row 24 Spare Message German' | French: 'S2 238 Row 24 Spare Message French'
  239 = 'S2 239 Row 24 Spare Message Default' | German: 'S2 239 Row 24 Spare Message German' | French: 'S2 239 Row 24 Spare Message French'
  240 = 'S2 240 Row 25 Failed To Advance.. Check Qxxx.x Default' | German: 'S2 240 Row 25 Failed To Advance.. Check Qxxx.x German' | French: 'S2 240 Row 25 Failed To Advance.. Check Qxxx.x French'
  241 = 'S2 241 Row 25 Failed To Return.. Check Qxxx.x Default' | German: 'S2 241 Row 25 Failed To Return.. Check Qxxx.x German' | French: 'S2 241 Row 25 Failed To Return.. Check Qxxx.x French'
  242 = 'S2 242 Row 25 Lost Advance Position... Check Ixxx.x Default' | German: 'S2 242 Row 25 Lost Advance Position... Check Ixxx.x German' | French: 'S2 242 Row 25 Lost Advance Position... Check Ixxx.x French'
  243 = 'S2 243 Row 25 Lost Return Position... Check Ixxx.x Default' | German: 'S2 243 Row 25 Lost Return Position... Check Ixxx.x German' | French: 'S2 243 Row 25 Lost Return Position... Check Ixxx.x French'
  244 = 'S2 244 Row 25 Switch Fault... Check Ixxx.x / Ixxx.x Default' | German: 'S2 244 Row 25 Switch Fault... Check Ixxx.x / Ixxx.x German' | French: 'S2 244 Row 25 Switch Fault... Check Ixxx.x / Ixxx.x French'
  245 = 'S2 245 Row 25 Spare Message Default' | German: 'S2 245 Row 25 Spare Message German' | French: 'S2 245 Row 25 Spare Message French'
  246 = 'S2 246 Row 25 Spare Message Default' | German: 'S2 246 Row 25 Spare Message German' | French: 'S2 246 Row 25 Spare Message French'
  247 = 'S2 247 Row 25 Spare Message Default' | German: 'S2 247 Row 25 Spare Message German' | French: 'S2 247 Row 25 Spare Message French'
  248 = 'S2 248 Row 25 Spare Message Default' | German: 'S2 248 Row 25 Spare Message German' | French: 'S2 248 Row 25 Spare Message French'
  249 = 'S2 249 Row 25 Spare Message Default' | German: 'S2 249 Row 25 Spare Message German' | French: 'S2 249 Row 25 Spare Message French'
  250 = 'S2 250 Row 26 Failed To Advance.. Check Qxxx.x Default' | German: 'S2 250 Row 26 Failed To Advance.. Check Qxxx.x German' | French: 'S2 250 Row 26 Failed To Advance.. Check Qxxx.x French'
  251 = 'S2 251 Row 26 Failed To Return.. Check Qxxx.x Default' | German: 'S2 251 Row 26 Failed To Return.. Check Qxxx.x German' | French: 'S2 251 Row 26 Failed To Return.. Check Qxxx.x French'
  252 = 'S2 252 Row 26 Lost Advance Position... Check Ixxx.x Default' | German: 'S2 252 Row 26 Lost Advance Position... Check Ixxx.x German' | French: 'S2 252 Row 26 Lost Advance Position... Check Ixxx.x French'
  253 = 'S2 253 Row 26 Lost Return Position... Check Ixxx.x Default' | German: 'S2 253 Row 26 Lost Return Position... Check Ixxx.x German' | French: 'S2 253 Row 26 Lost Return Position... Check Ixxx.x French'
  254 = 'S2 254 Row 26 Switch Fault... Check Ixxx.x / Ixxx.x Default' | German: 'S2 254 Row 26 Switch Fault... Check Ixxx.x / Ixxx.x German' | French: 'S2 254 Row 26 Switch Fault... Check Ixxx.x / Ixxx.x French'
  255 = 'S2 255 Row 26 Spare Message Default' | German: 'S2 255 Row 26 Spare Message German' | French: 'S2 255 Row 26 Spare Message French'
  256 = 'S2 256 Row 26 Spare Message Default' | German: 'S2 256 Row 26 Spare Message German' | French: 'S2 256 Row 26 Spare Message French'
  257 = 'S2 257 Row 26 Spare Message Default' | German: 'S2 257 Row 26 Spare Message German' | French: 'S2 257 Row 26 Spare Message French'
  258 = 'S2 258 Row 26 Spare Message Default' | German: 'S2 258 Row 26 Spare Message German' | French: 'S2 258 Row 26 Spare Message French'
  259 = 'S2 259 Row 26 Spare Message Default' | German: 'S2 259 Row 26 Spare Message German' | French: 'S2 259 Row 26 Spare Message French'
  260 = 'S2 260 Row 27 Failed To Advance.. Check Qxxx.x Default' | German: 'S2 260 Row 27 Failed To Advance.. Check Qxxx.x German' | French: 'S2 260 Row 27 Failed To Advance.. Check Qxxx.x French'
  261 = 'S2 261 Row 27 Failed To Return.. Check Qxxx.x Default' | German: 'S2 261 Row 27 Failed To Return.. Check Qxxx.x German' | French: 'S2 261 Row 27 Failed To Return.. Check Qxxx.x French'
  262 = 'S2 262 Row 27 Lost Advance Position... Check Ixxx.x Default' | German: 'S2 262 Row 27 Lost Advance Position... Check Ixxx.x German' | French: 'S2 262 Row 27 Lost Advance Position... Check Ixxx.x French'
  263 = 'S2 263 Row 27 Lost Return Position... Check Ixxx.x Default' | German: 'S2 263 Row 27 Lost Return Position... Check Ixxx.x German' | French: 'S2 263 Row 27 Lost Return Position... Check Ixxx.x French'
  264 = 'S2 264 Row 27 Switch Fault... Check Ixxx.x / Ixxx.x Default' | German: 'S2 264 Row 27 Switch Fault... Check Ixxx.x / Ixxx.x German' | French: 'S2 264 Row 27 Switch Fault... Check Ixxx.x / Ixxx.x French'
  265 = 'S2 265 Row 27 Spare Message Default' | German: 'S2 265 Row 27 Spare Message German' | French: 'S2 265 Row 27 Spare Message French'
  266 = 'S2 266 Row 27 Spare Message Default' | German: 'S2 266 Row 27 Spare Message German' | French: 'S2 266 Row 27 Spare Message French'
  267 = 'S2 267 Row 27 Spare Message Default' | German: 'S2 267 Row 27 Spare Message German' | French: 'S2 267 Row 27 Spare Message French'
  268 = 'S2 268 Row 27 Spare Message Default' | German: 'S2 268 Row 27 Spare Message German' | French: 'S2 268 Row 27 Spare Message French'
  269 = 'S2 269 Row 27 Spare Message Default' | German: 'S2 269 Row 27 Spare Message German' | French: 'S2 269 Row 27 Spare Message French'
  270 = 'S2 270 Row 28 Failed To Advance.. Check Qxxx.x Default' | German: 'S2 270 Row 28 Failed To Advance.. Check Qxxx.x German' | French: 'S2 270 Row 28 Failed To Advance.. Check Qxxx.x French'
  271 = 'S2 271 Row 28 Failed To Return.. Check Qxxx.x Default' | German: 'S2 271 Row 28 Failed To Return.. Check Qxxx.x German' | French: 'S2 271 Row 28 Failed To Return.. Check Qxxx.x French'
  272 = 'S2 272 Row 28 Lost Advance Position... Check Ixxx.x Default' | German: 'S2 272 Row 28 Lost Advance Position... Check Ixxx.x German' | French: 'S2 272 Row 28 Lost Advance Position... Check Ixxx.x French'
  273 = 'S2 273 Row 28 Lost Return Position... Check Ixxx.x Default' | German: 'S2 273 Row 28 Lost Return Position... Check Ixxx.x German' | French: 'S2 273 Row 28 Lost Return Position... Check Ixxx.x French'
  274 = 'S2 274 Row 28 Switch Fault... Check Ixxx.x / Ixxx.x Default' | German: 'S2 274 Row 28 Switch Fault... Check Ixxx.x / Ixxx.x German' | French: 'S2 274 Row 28 Switch Fault... Check Ixxx.x / Ixxx.x French'
  275 = 'S2 275 Row 28 Spare Message Default' | German: 'S2 275 Row 28 Spare Message German' | French: 'S2 275 Row 28 Spare Message French'
  276 = 'S2 276 Row 28 Spare Message Default' | German: 'S2 276 Row 28 Spare Message German' | French: 'S2 276 Row 28 Spare Message French'
  277 = 'S2 277 Row 28 Spare Message Default' | German: 'S2 277 Row 28 Spare Message German' | French: 'S2 277 Row 28 Spare Message French'
  278 = 'S2 278 Row 28 Spare Message Default' | German: 'S2 278 Row 28 Spare Message German' | French: 'S2 278 Row 28 Spare Message French'
  279 = 'S2 279 Row 28 Spare Message Default' | German: 'S2 279 Row 28 Spare Message German' | French: 'S2 279 Row 28 Spare Message French'
  280 = 'S2 280 Row 29 Failed To Advance.. Check Qxxx.x Default' | German: 'S2 280 Row 29 Failed To Advance.. Check Qxxx.x German' | French: 'S2 280 Row 29 Failed To Advance.. Check Qxxx.x French'
  281 = 'S2 281 Row 29 Failed To Return.. Check Qxxx.x Default' | German: 'S2 281 Row 29 Failed To Return.. Check Qxxx.x German' | French: 'S2 281 Row 29 Failed To Return.. Check Qxxx.x French'
  282 = 'S2 282 Row 29 Lost Advance Position... Check Ixxx.x Default' | German: 'S2 282 Row 29 Lost Advance Position... Check Ixxx.x German' | French: 'S2 282 Row 29 Lost Advance Position... Check Ixxx.x French'
  283 = 'S2 283 Row 29 Lost Return Position... Check Ixxx.x Default' | German: 'S2 283 Row 29 Lost Return Position... Check Ixxx.x German' | French: 'S2 283 Row 29 Lost Return Position... Check Ixxx.x French'
  284 = 'S2 284 Row 29 Switch Fault... Check Ixxx.x / Ixxx.x Default' | German: 'S2 284 Row 29 Switch Fault... Check Ixxx.x / Ixxx.x German' | French: 'S2 284 Row 29 Switch Fault... Check Ixxx.x / Ixxx.x French'
  285 = 'S2 285 Row 29 Spare Message Default' | German: 'S2 285 Row 29 Spare Message German' | French: 'S2 285 Row 29 Spare Message French'
  286 = 'S2 286 Row 29 Spare Message Default' | German: 'S2 286 Row 29 Spare Message German' | French: 'S2 286 Row 29 Spare Message French'
  287 = 'S2 287 Row 29 Spare Message Default' | German: 'S2 287 Row 29 Spare Message German' | French: 'S2 287 Row 29 Spare Message French'
  288 = 'S2 288 Row 29 Spare Message Default' | German: 'S2 288 Row 29 Spare Message German' | French: 'S2 288 Row 29 Spare Message French'
  289 = 'S2 289 Row 29 Spare Message Default' | German: 'S2 289 Row 29 Spare Message German' | French: 'S2 289 Row 29 Spare Message French'
  290 = 'S2 290 Row 30 Failed To Advance.. Check Qxxx.x Default' | German: 'S2 290 Row 30 Failed To Advance.. Check Qxxx.x German' | French: 'S2 290 Row 30 Failed To Advance.. Check Qxxx.x French'
  291 = 'S2 291 Row 30 Failed To Return.. Check Qxxx.x Default' | German: 'S2 291 Row 30 Failed To Return.. Check Qxxx.x German' | French: 'S2 291 Row 30 Failed To Return.. Check Qxxx.x French'
  292 = 'S2 292 Row 30 Lost Advance Position... Check Ixxx.x Default' | German: 'S2 292 Row 30 Lost Advance Position... Check Ixxx.x German' | French: 'S2 292 Row 30 Lost Advance Position... Check Ixxx.x French'
  293 = 'S2 293 Row 30 Lost Return Position... Check Ixxx.x Default' | German: 'S2 293 Row 30 Lost Return Position... Check Ixxx.x German' | French: 'S2 293 Row 30 Lost Return Position... Check Ixxx.x French'
  294 = 'S2 294 Row 30 Switch Fault... Check Ixxx.x / Ixxx.x Default' | German: 'S2 294 Row 30 Switch Fault... Check Ixxx.x / Ixxx.x German' | French: 'S2 294 Row 30 Switch Fault... Check Ixxx.x / Ixxx.x French'
  295 = 'S2 295 Row 30 Spare Message Default' | German: 'S2 295 Row 30 Spare Message German' | French: 'S2 295 Row 30 Spare Message French'
  296 = 'S2 296 Row 30 Spare Message Default' | German: 'S2 296 Row 30 Spare Message German' | French: 'S2 296 Row 30 Spare Message French'
  297 = 'S2 297 Row 30 Spare Message Default' | German: 'S2 297 Row 30 Spare Message German' | French: 'S2 297 Row 30 Spare Message French'
  298 = 'S2 298 Row 30 Spare Message Default' | German: 'S2 298 Row 30 Spare Message German' | French: 'S2 298 Row 30 Spare Message French'
  299 = 'S2 299 Row 30 Spare Message Default' | German: 'S2 299 Row 30 Spare Message German' | French: 'S2 299 Row 30 Spare Message French'
  300 = 'S2 300 Row 31 Failed To Advance.. Check Qxxx.x Default' | German: 'S2 300 Row 31 Failed To Advance.. Check Qxxx.x German' | French: 'S2 300 Row 31 Failed To Advance.. Check Qxxx.x French'
  301 = 'S2 301 Row 31 Failed To Return.. Check Qxxx.x Default' | German: 'S2 301 Row 31 Failed To Return.. Check Qxxx.x German' | French: 'S2 301 Row 31 Failed To Return.. Check Qxxx.x French'
  302 = 'S2 302 Row 31 Lost Advance Position... Check Ixxx.x Default' | German: 'S2 302 Row 31 Lost Advance Position... Check Ixxx.x German' | French: 'S2 302 Row 31 Lost Advance Position... Check Ixxx.x French'
  303 = 'S2 303 Row 31 Lost Return Position... Check Ixxx.x Default' | German: 'S2 303 Row 31 Lost Return Position... Check Ixxx.x German' | French: 'S2 303 Row 31 Lost Return Position... Check Ixxx.x French'
  304 = 'S2 304 Row 31 Switch Fault... Check Ixxx.x / Ixxx.x Default' | German: 'S2 304 Row 31 Switch Fault... Check Ixxx.x / Ixxx.x German' | French: 'S2 304 Row 31 Switch Fault... Check Ixxx.x / Ixxx.x French'
  305 = 'S2 305 Row 31 Spare Message Default' | German: 'S2 305 Row 31 Spare Message German' | French: 'S2 305 Row 31 Spare Message French'
  306 = 'S2 306 Row 31 Spare Message Default' | German: 'S2 306 Row 31 Spare Message German' | French: 'S2 306 Row 31 Spare Message French'
  307 = 'S2 307 Row 31 Spare Message Default' | German: 'S2 307 Row 31 Spare Message German' | French: 'S2 307 Row 31 Spare Message French'
  308 = 'S2 308 Row 31 Spare Message Default' | German: 'S2 308 Row 31 Spare Message German' | French: 'S2 308 Row 31 Spare Message French'
  309 = 'S2 309 Row 31 Spare Message Default' | German: 'S2 309 Row 31 Spare Message German' | French: 'S2 309 Row 31 Spare Message French'
  310 = 'S2 310 Row 32 Failed To Advance.. Check Qxxx.x Default' | German: 'S2 310 Row 32 Failed To Advance.. Check Qxxx.x German' | French: 'S2 310 Row 32 Failed To Advance.. Check Qxxx.x French'
  311 = 'S2 311 Row 32 Failed To Return.. Check Qxxx.x Default' | German: 'S2 311 Row 32 Failed To Return.. Check Qxxx.x German' | French: 'S2 311 Row 32 Failed To Return.. Check Qxxx.x French'
  312 = 'S2 312 Row 32 Lost Advance Position... Check Ixxx.x Default' | German: 'S2 312 Row 32 Lost Advance Position... Check Ixxx.x German' | French: 'S2 312 Row 32 Lost Advance Position... Check Ixxx.x French'
  313 = 'S2 313 Row 32 Lost Return Position... Check Ixxx.x Default' | German: 'S2 313 Row 32 Lost Return Position... Check Ixxx.x German' | French: 'S2 313 Row 32 Lost Return Position... Check Ixxx.x French'
  314 = 'S2 314 Row 32 Switch Fault... Check Ixxx.x / Ixxx.x Default' | German: 'S2 314 Row 32 Switch Fault... Check Ixxx.x / Ixxx.x German' | French: 'S2 314 Row 32 Switch Fault... Check Ixxx.x / Ixxx.x French'
  315 = 'S2 315 Row 32 Spare Message Default' | German: 'S2 315 Row 32 Spare Message German' | French: 'S2 315 Row 32 Spare Message French'
  316 = 'S2 316 Row 32 Spare Message Default' | German: 'S2 316 Row 32 Spare Message German' | French: 'S2 316 Row 32 Spare Message French'
  317 = 'S2 317 Row 32 Spare Message Default' | German: 'S2 317 Row 32 Spare Message German' | French: 'S2 317 Row 32 Spare Message French'
  318 = 'S2 318 Row 32 Spare Message Default' | German: 'S2 318 Row 32 Spare Message German' | French: 'S2 318 Row 32 Spare Message French'
  319 = 'S2 319 Row 32 Spare Message Default' | German: 'S2 319 Row 32 Spare Message German' | French: 'S2 319 Row 32 Spare Message French'
  320 = 'S2 320 Row 33 Failed To Advance.. Check Qxxx.x Default' | German: 'S2 320 Row 33 Failed To Advance.. Check Qxxx.x German' | French: 'S2 320 Row 33 Failed To Advance.. Check Qxxx.x French'
  321 = 'S2 321 Row 33 Failed To Return.. Check Qxxx.x Default' | German: 'S2 321 Row 33 Failed To Return.. Check Qxxx.x German' | French: 'S2 321 Row 33 Failed To Return.. Check Qxxx.x French'
  322 = 'S2 322 Row 33 Lost Advance Position... Check Ixxx.x Default' | German: 'S2 322 Row 33 Lost Advance Position... Check Ixxx.x German' | French: 'S2 322 Row 33 Lost Advance Position... Check Ixxx.x French'
  323 = 'S2 323 Row 33 Lost Return Position... Check Ixxx.x Default' | German: 'S2 323 Row 33 Lost Return Position... Check Ixxx.x German' | French: 'S2 323 Row 33 Lost Return Position... Check Ixxx.x French'
  324 = 'S2 324 Row 33 Switch Fault... Check Ixxx.x / Ixxx.x Default' | German: 'S2 324 Row 33 Switch Fault... Check Ixxx.x / Ixxx.x German' | French: 'S2 324 Row 33 Switch Fault... Check Ixxx.x / Ixxx.x French'
  325 = 'S2 325 Row 33 Spare Message Default' | German: 'S2 325 Row 33 Spare Message German' | French: 'S2 325 Row 33 Spare Message French'
  326 = 'S2 326 Row 33 Spare Message Default' | German: 'S2 326 Row 33 Spare Message German' | French: 'S2 326 Row 33 Spare Message French'
  327 = 'S2 327 Row 33 Spare Message Default' | German: 'S2 327 Row 33 Spare Message German' | French: 'S2 327 Row 33 Spare Message French'
  328 = 'S2 328 Row 33 Spare Message Default' | German: 'S2 328 Row 33 Spare Message German' | French: 'S2 328 Row 33 Spare Message French'
  329 = 'S2 329 Row 33 Spare Message Default' | German: 'S2 329 Row 33 Spare Message German' | French: 'S2 329 Row 33 Spare Message French'
  330 = 'S2 330 Row 34 Failed To Advance.. Check Qxxx.x Default' | German: 'S2 330 Row 34 Failed To Advance.. Check Qxxx.x German' | French: 'S2 330 Row 34 Failed To Advance.. Check Qxxx.x French'
  331 = 'S2 331 Row 34 Failed To Return.. Check Qxxx.x Default' | German: 'S2 331 Row 34 Failed To Return.. Check Qxxx.x German' | French: 'S2 331 Row 34 Failed To Return.. Check Qxxx.x French'
  332 = 'S2 332 Row 34 Lost Advance Position... Check Ixxx.x Default' | German: 'S2 332 Row 34 Lost Advance Position... Check Ixxx.x German' | French: 'S2 332 Row 34 Lost Advance Position... Check Ixxx.x French'
  333 = 'S2 333 Row 34 Lost Return Position... Check Ixxx.x Default' | German: 'S2 333 Row 34 Lost Return Position... Check Ixxx.x German' | French: 'S2 333 Row 34 Lost Return Position... Check Ixxx.x French'
  334 = 'S2 334 Row 34 Switch Fault... Check Ixxx.x / Ixxx.x Default' | German: 'S2 334 Row 34 Switch Fault... Check Ixxx.x / Ixxx.x German' | French: 'S2 334 Row 34 Switch Fault... Check Ixxx.x / Ixxx.x French'
  335 = 'S2 335 Row 34 Spare Message Default' | German: 'S2 335 Row 34 Spare Message German' | French: 'S2 335 Row 34 Spare Message French'
  336 = 'S2 336 Row 34 Spare Message Default' | German: 'S2 336 Row 34 Spare Message German' | French: 'S2 336 Row 34 Spare Message French'
  337 = 'S2 337 Row 34 Spare Message Default' | German: 'S2 337 Row 34 Spare Message German' | French: 'S2 337 Row 34 Spare Message French'
  338 = 'S2 338 Row 34 Spare Message Default' | German: 'S2 338 Row 34 Spare Message German' | French: 'S2 338 Row 34 Spare Message French'
  339 = 'S2 339 Row 34 Spare Message Default' | German: 'S2 339 Row 34 Spare Message German' | French: 'S2 339 Row 34 Spare Message French'
  340 = 'S2 340 Row 35 Failed To Advance.. Check Qxxx.x Default' | German: 'S2 340 Row 35 Failed To Advance.. Check Qxxx.x German' | French: 'S2 340 Row 35 Failed To Advance.. Check Qxxx.x French'
  341 = 'S2 341 Row 35 Failed To Return.. Check Qxxx.x Default' | German: 'S2 341 Row 35 Failed To Return.. Check Qxxx.x German' | French: 'S2 341 Row 35 Failed To Return.. Check Qxxx.x French'
  342 = 'S2 342 Row 35 Lost Advance Position... Check Ixxx.x Default' | German: 'S2 342 Row 35 Lost Advance Position... Check Ixxx.x German' | French: 'S2 342 Row 35 Lost Advance Position... Check Ixxx.x French'
  343 = 'S2 343 Row 35 Lost Return Position... Check Ixxx.x Default' | German: 'S2 343 Row 35 Lost Return Position... Check Ixxx.x German' | French: 'S2 343 Row 35 Lost Return Position... Check Ixxx.x French'
  344 = 'S2 344 Row 35 Switch Fault... Check Ixxx.x / Ixxx.x Default' | German: 'S2 344 Row 35 Switch Fault... Check Ixxx.x / Ixxx.x German' | French: 'S2 344 Row 35 Switch Fault... Check Ixxx.x / Ixxx.x French'
  345 = 'S2 345 Row 35 Spare Message Default' | German: 'S2 345 Row 35 Spare Message German' | French: 'S2 345 Row 35 Spare Message French'
  346 = 'S2 346 Row 35 Spare Message Default' | German: 'S2 346 Row 35 Spare Message German' | French: 'S2 346 Row 35 Spare Message French'
  347 = 'S2 347 Row 35 Spare Message Default' | German: 'S2 347 Row 35 Spare Message German' | French: 'S2 347 Row 35 Spare Message French'
  348 = 'S2 348 Row 35 Spare Message Default' | German: 'S2 348 Row 35 Spare Message German' | French: 'S2 348 Row 35 Spare Message French'
  349 = 'S2 349 Row 35 Spare Message Default' | German: 'S2 349 Row 35 Spare Message German' | French: 'S2 349 Row 35 Spare Message French'
  350 = 'S2 350 Row 36 Failed To Advance.. Check Qxxx.x Default' | German: 'S2 350 Row 36 Failed To Advance.. Check Qxxx.x German' | French: 'S2 350 Row 36 Failed To Advance.. Check Qxxx.x French'
  351 = 'S2 351 Row 36 Failed To Return.. Check Qxxx.x Default' | German: 'S2 351 Row 36 Failed To Return.. Check Qxxx.x German' | French: 'S2 351 Row 36 Failed To Return.. Check Qxxx.x French'
  352 = 'S2 352 Row 36 Lost Advance Position... Check Ixxx.x Default' | German: 'S2 352 Row 36 Lost Advance Position... Check Ixxx.x German' | French: 'S2 352 Row 36 Lost Advance Position... Check Ixxx.x French'
  353 = 'S2 353 Row 36 Lost Return Position... Check Ixxx.x Default' | German: 'S2 353 Row 36 Lost Return Position... Check Ixxx.x German' | French: 'S2 353 Row 36 Lost Return Position... Check Ixxx.x French'
  354 = 'S2 354 Row 36 Switch Fault... Check Ixxx.x / Ixxx.x Default' | German: 'S2 354 Row 36 Switch Fault... Check Ixxx.x / Ixxx.x German' | French: 'S2 354 Row 36 Switch Fault... Check Ixxx.x / Ixxx.x French'
  355 = 'S2 355 Row 36 Spare Message Default' | German: 'S2 355 Row 36 Spare Message German' | French: 'S2 355 Row 36 Spare Message French'
  356 = 'S2 356 Row 36 Spare Message Default' | German: 'S2 356 Row 36 Spare Message German' | French: 'S2 356 Row 36 Spare Message French'
  357 = 'S2 357 Row 36 Spare Message Default' | German: 'S2 357 Row 36 Spare Message German' | French: 'S2 357 Row 36 Spare Message French'
  358 = 'S2 358 Row 36 Spare Message Default' | German: 'S2 358 Row 36 Spare Message German' | French: 'S2 358 Row 36 Spare Message French'
  359 = 'S2 359 Row 36 Spare Message Default' | German: 'S2 359 Row 36 Spare Message German' | French: 'S2 359 Row 36 Spare Message French'
  360 = 'S2 360 Row 37 Failed To Advance.. Check Qxxx.x Default' | German: 'S2 360 Row 37 Failed To Advance.. Check Qxxx.x German' | French: 'S2 360 Row 37 Failed To Advance.. Check Qxxx.x French'
  361 = 'S2 361 Row 37 Failed To Return.. Check Qxxx.x Default' | German: 'S2 361 Row 37 Failed To Return.. Check Qxxx.x German' | French: 'S2 361 Row 37 Failed To Return.. Check Qxxx.x French'
  362 = 'S2 362 Row 37 Lost Advance Position... Check Ixxx.x Default' | German: 'S2 362 Row 37 Lost Advance Position... Check Ixxx.x German' | French: 'S2 362 Row 37 Lost Advance Position... Check Ixxx.x French'
  363 = 'S2 363 Row 37 Lost Return Position... Check Ixxx.x Default' | German: 'S2 363 Row 37 Lost Return Position... Check Ixxx.x German' | French: 'S2 363 Row 37 Lost Return Position... Check Ixxx.x French'
  364 = 'S2 364 Row 37 Switch Fault... Check Ixxx.x / Ixxx.x Default' | German: 'S2 364 Row 37 Switch Fault... Check Ixxx.x / Ixxx.x German' | French: 'S2 364 Row 37 Switch Fault... Check Ixxx.x / Ixxx.x French'
  365 = 'S2 365 Row 37 Spare Message Default' | German: 'S2 365 Row 37 Spare Message German' | French: 'S2 365 Row 37 Spare Message French'
  366 = 'S2 366 Row 37 Spare Message Default' | German: 'S2 366 Row 37 Spare Message German' | French: 'S2 366 Row 37 Spare Message French'
  367 = 'S2 367 Row 37 Spare Message Default' | German: 'S2 367 Row 37 Spare Message German' | French: 'S2 367 Row 37 Spare Message French'
  368 = 'S2 368 Row 37 Spare Message Default' | German: 'S2 368 Row 37 Spare Message German' | French: 'S2 368 Row 37 Spare Message French'
  369 = 'S2 369 Row 37 Spare Message Default' | German: 'S2 369 Row 37 Spare Message German' | French: 'S2 369 Row 37 Spare Message French'
  370 = 'S2 370 Row 38 Failed To Advance.. Check Qxxx.x Default' | German: 'S2 370 Row 38 Failed To Advance.. Check Qxxx.x German' | French: 'S2 370 Row 38 Failed To Advance.. Check Qxxx.x French'
  371 = 'S2 371 Row 38 Failed To Return.. Check Qxxx.x Default' | German: 'S2 371 Row 38 Failed To Return.. Check Qxxx.x German' | French: 'S2 371 Row 38 Failed To Return.. Check Qxxx.x French'
  372 = 'S2 372 Row 38 Lost Advance Position... Check Ixxx.x Default' | German: 'S2 372 Row 38 Lost Advance Position... Check Ixxx.x German' | French: 'S2 372 Row 38 Lost Advance Position... Check Ixxx.x French'
  373 = 'S2 373 Row 38 Lost Return Position... Check Ixxx.x Default' | German: 'S2 373 Row 38 Lost Return Position... Check Ixxx.x German' | French: 'S2 373 Row 38 Lost Return Position... Check Ixxx.x French'
  374 = 'S2 374 Row 38 Switch Fault... Check Ixxx.x / Ixxx.x Default' | German: 'S2 374 Row 38 Switch Fault... Check Ixxx.x / Ixxx.x German' | French: 'S2 374 Row 38 Switch Fault... Check Ixxx.x / Ixxx.x French'
  375 = 'S2 375 Row 38 Spare Message Default' | German: 'S2 375 Row 38 Spare Message German' | French: 'S2 375 Row 38 Spare Message French'
  376 = 'S2 376 Row 38 Spare Message Default' | German: 'S2 376 Row 38 Spare Message German' | French: 'S2 376 Row 38 Spare Message French'
  377 = 'S2 377 Row 38 Spare Message Default' | German: 'S2 377 Row 38 Spare Message German' | French: 'S2 377 Row 38 Spare Message French'
  378 = 'S2 378 Row 38 Spare Message Default' | German: 'S2 378 Row 38 Spare Message German' | French: 'S2 378 Row 38 Spare Message French'
  379 = 'S2 379 Row 38 Spare Message Default' | German: 'S2 379 Row 38 Spare Message German' | French: 'S2 379 Row 38 Spare Message French'
  380 = 'S2 380 Row 39 Failed To Advance.. Check Qxxx.x Default' | German: 'S2 380 Row 39 Failed To Advance.. Check Qxxx.x German' | French: 'S2 380 Row 39 Failed To Advance.. Check Qxxx.x French'
  381 = 'S2 381 Row 39 Failed To Return.. Check Qxxx.x Default' | German: 'S2 381 Row 39 Failed To Return.. Check Qxxx.x German' | French: 'S2 381 Row 39 Failed To Return.. Check Qxxx.x French'
  382 = 'S2 382 Row 39 Lost Advance Position... Check Ixxx.x Default' | German: 'S2 382 Row 39 Lost Advance Position... Check Ixxx.x German' | French: 'S2 382 Row 39 Lost Advance Position... Check Ixxx.x French'
  383 = 'S2 383 Row 39 Lost Return Position... Check Ixxx.x Default' | German: 'S2 383 Row 39 Lost Return Position... Check Ixxx.x German' | French: 'S2 383 Row 39 Lost Return Position... Check Ixxx.x French'
  384 = 'S2 384 Row 39 Switch Fault... Check Ixxx.x / Ixxx.x Default' | German: 'S2 384 Row 39 Switch Fault... Check Ixxx.x / Ixxx.x German' | French: 'S2 384 Row 39 Switch Fault... Check Ixxx.x / Ixxx.x French'
  385 = 'S2 385 Row 39 Spare Message Default' | German: 'S2 385 Row 39 Spare Message German' | French: 'S2 385 Row 39 Spare Message French'
  386 = 'S2 386 Row 39 Spare Message Default' | German: 'S2 386 Row 39 Spare Message German' | French: 'S2 386 Row 39 Spare Message French'
  387 = 'S2 387 Row 39 Spare Message Default' | German: 'S2 387 Row 39 Spare Message German' | French: 'S2 387 Row 39 Spare Message French'
  388 = 'S2 388 Row 39 Spare Message Default' | German: 'S2 388 Row 39 Spare Message German' | French: 'S2 388 Row 39 Spare Message French'
  389 = 'S2 389 Row 39 Spare Message Default' | German: 'S2 389 Row 39 Spare Message German' | French: 'S2 389 Row 39 Spare Message French'
  390 = 'S2 390 Row 40 Failed To Advance.. Check Qxxx.x Default' | German: 'S2 390 Row 40 Failed To Advance.. Check Qxxx.x German' | French: 'S2 390 Row 40 Failed To Advance.. Check Qxxx.x French'
  391 = 'S2 391 Row 40 Failed To Return.. Check Qxxx.x Default' | German: 'S2 391 Row 40 Failed To Return.. Check Qxxx.x German' | French: 'S2 391 Row 40 Failed To Return.. Check Qxxx.x French'
  392 = 'S2 392 Row 40 Lost Advance Position... Check Ixxx.x Default' | German: 'S2 392 Row 40 Lost Advance Position... Check Ixxx.x German' | French: 'S2 392 Row 40 Lost Advance Position... Check Ixxx.x French'
  393 = 'S2 393 Row 40 Lost Return Position... Check Ixxx.x Default' | German: 'S2 393 Row 40 Lost Return Position... Check Ixxx.x German' | French: 'S2 393 Row 40 Lost Return Position... Check Ixxx.x French'
  394 = 'S2 394 Row 40 Switch Fault... Check Ixxx.x / Ixxx.x Default' | German: 'S2 394 Row 40 Switch Fault... Check Ixxx.x / Ixxx.x German' | French: 'S2 394 Row 40 Switch Fault... Check Ixxx.x / Ixxx.x French'
  395 = 'S2 395 Row 40 Spare Message Default' | German: 'S2 395 Row 40 Spare Message German' | French: 'S2 395 Row 40 Spare Message French'
  396 = 'S2 396 Row 40 Spare Message Default' | German: 'S2 396 Row 40 Spare Message German' | French: 'S2 396 Row 40 Spare Message French'
  397 = 'S2 397 Row 40 Spare Message Default' | German: 'S2 397 Row 40 Spare Message German' | French: 'S2 397 Row 40 Spare Message French'
  398 = 'S2 398 Row 40 Spare Message Default' | German: 'S2 398 Row 40 Spare Message German' | French: 'S2 398 Row 40 Spare Message French'
  399 = 'S2 399 Row 40 Spare Message Default' | German: 'S2 399 Row 40 Spare Message German' | French: 'S2 399 Row 40 Spare Message French'
  400 = 'S2 400 Row 41 Failed To Advance.. Check Qxxx.x Default' | German: 'S2 400 Row 41 Failed To Advance.. Check Qxxx.x German' | French: 'S2 400 Row 41 Failed To Advance.. Check Qxxx.x French'
  401 = 'S2 401 Row 41 Failed To Return.. Check Qxxx.x Default' | German: 'S2 401 Row 41 Failed To Return.. Check Qxxx.x German' | French: 'S2 401 Row 41 Failed To Return.. Check Qxxx.x French'
  402 = 'S2 402 Row 41 Lost Advance Position... Check Ixxx.x Default' | German: 'S2 402 Row 41 Lost Advance Position... Check Ixxx.x German' | French: 'S2 402 Row 41 Lost Advance Position... Check Ixxx.x French'
  403 = 'S2 403 Row 41 Lost Return Position... Check Ixxx.x Default' | German: 'S2 403 Row 41 Lost Return Position... Check Ixxx.x German' | French: 'S2 403 Row 41 Lost Return Position... Check Ixxx.x French'
  404 = 'S2 404 Row 41 Switch Fault... Check Ixxx.x / Ixxx.x Default' | German: 'S2 404 Row 41 Switch Fault... Check Ixxx.x / Ixxx.x German' | French: 'S2 404 Row 41 Switch Fault... Check Ixxx.x / Ixxx.x French'
  405 = 'S2 405 Row 41 Spare Message Default' | German: 'S2 405 Row 41 Spare Message German' | French: 'S2 405 Row 41 Spare Message French'
  406 = 'S2 406 Row 41 Spare Message Default' | German: 'S2 406 Row 41 Spare Message German' | French: 'S2 406 Row 41 Spare Message French'
  407 = 'S2 407 Row 41 Spare Message Default' | German: 'S2 407 Row 41 Spare Message German' | French: 'S2 407 Row 41 Spare Message French'
  408 = 'S2 408 Row 41 Spare Message Default' | German: 'S2 408 Row 41 Spare Message German' | French: 'S2 408 Row 41 Spare Message French'
  409 = 'S2 409 Row 41 Spare Message Default' | German: 'S2 409 Row 41 Spare Message German' | French: 'S2 409 Row 41 Spare Message French'
  410 = 'S2 410 Row 42 Failed To Advance.. Check Qxxx.x Default' | German: 'S2 410 Row 42 Failed To Advance.. Check Qxxx.x German' | French: 'S2 410 Row 42 Failed To Advance.. Check Qxxx.x French'
  411 = 'S2 411 Row 42 Failed To Return.. Check Qxxx.x Default' | German: 'S2 411 Row 42 Failed To Return.. Check Qxxx.x German' | French: 'S2 411 Row 42 Failed To Return.. Check Qxxx.x French'
  412 = 'S2 412 Row 42 Lost Advance Position... Check Ixxx.x Default' | German: 'S2 412 Row 42 Lost Advance Position... Check Ixxx.x German' | French: 'S2 412 Row 42 Lost Advance Position... Check Ixxx.x French'
  413 = 'S2 413 Row 42 Lost Return Position... Check Ixxx.x Default' | German: 'S2 413 Row 42 Lost Return Position... Check Ixxx.x German' | French: 'S2 413 Row 42 Lost Return Position... Check Ixxx.x French'
  414 = 'S2 414 Row 42 Switch Fault... Check Ixxx.x / Ixxx.x Default' | German: 'S2 414 Row 42 Switch Fault... Check Ixxx.x / Ixxx.x German' | French: 'S2 414 Row 42 Switch Fault... Check Ixxx.x / Ixxx.x French'
  415 = 'S2 415 Row 42 Spare Message Default' | German: 'S2 415 Row 42 Spare Message German' | French: 'S2 415 Row 42 Spare Message French'
  416 = 'S2 416 Row 42 Spare Message Default' | German: 'S2 416 Row 42 Spare Message German' | French: 'S2 416 Row 42 Spare Message French'
  417 = 'S2 417 Row 42 Spare Message Default' | German: 'S2 417 Row 42 Spare Message German' | French: 'S2 417 Row 42 Spare Message French'
  418 = 'S2 418 Row 42 Spare Message Default' | German: 'S2 418 Row 42 Spare Message German' | French: 'S2 418 Row 42 Spare Message French'
  419 = 'S2 419 Row 42 Spare Message Default' | German: 'S2 419 Row 42 Spare Message German' | French: 'S2 419 Row 42 Spare Message French'
  420 = 'S2 420 Row 43 Failed To Advance.. Check Qxxx.x Default' | German: 'S2 420 Row 43 Failed To Advance.. Check Qxxx.x German' | French: 'S2 420 Row 43 Failed To Advance.. Check Qxxx.x French'
  421 = 'S2 421 Row 43 Failed To Return.. Check Qxxx.x Default' | German: 'S2 421 Row 43 Failed To Return.. Check Qxxx.x German' | French: 'S2 421 Row 43 Failed To Return.. Check Qxxx.x French'
  422 = 'S2 422 Row 43 Lost Advance Position... Check Ixxx.x Default' | German: 'S2 422 Row 43 Lost Advance Position... Check Ixxx.x German' | French: 'S2 422 Row 43 Lost Advance Position... Check Ixxx.x French'
  423 = 'S2 423 Row 43 Lost Return Position... Check Ixxx.x Default' | German: 'S2 423 Row 43 Lost Return Position... Check Ixxx.x German' | French: 'S2 423 Row 43 Lost Return Position... Check Ixxx.x French'
  424 = 'S2 424 Row 43 Switch Fault... Check Ixxx.x / Ixxx.x Default' | German: 'S2 424 Row 43 Switch Fault... Check Ixxx.x / Ixxx.x German' | French: 'S2 424 Row 43 Switch Fault... Check Ixxx.x / Ixxx.x French'
  425 = 'S2 425 Row 43 Spare Message Default' | German: 'S2 425 Row 43 Spare Message German' | French: 'S2 425 Row 43 Spare Message French'
  426 = 'S2 426 Row 43 Spare Message Default' | German: 'S2 426 Row 43 Spare Message German' | French: 'S2 426 Row 43 Spare Message French'
  427 = 'S2 427 Row 43 Spare Message Default' | German: 'S2 427 Row 43 Spare Message German' | French: 'S2 427 Row 43 Spare Message French'
  428 = 'S2 428 Row 43 Spare Message Default' | German: 'S2 428 Row 43 Spare Message German' | French: 'S2 428 Row 43 Spare Message French'
  429 = 'S2 429 Row 43 Spare Message Default' | German: 'S2 429 Row 43 Spare Message German' | French: 'S2 429 Row 43 Spare Message French'
  430 = 'S2 430 Row 44 Failed To Advance.. Check Qxxx.x Default' | German: 'S2 430 Row 44 Failed To Advance.. Check Qxxx.x German' | French: 'S2 430 Row 44 Failed To Advance.. Check Qxxx.x French'
  431 = 'S2 431 Row 44 Failed To Return.. Check Qxxx.x Default' | German: 'S2 431 Row 44 Failed To Return.. Check Qxxx.x German' | French: 'S2 431 Row 44 Failed To Return.. Check Qxxx.x French'
  432 = 'S2 432 Row 44 Lost Advance Position... Check Ixxx.x Default' | German: 'S2 432 Row 44 Lost Advance Position... Check Ixxx.x German' | French: 'S2 432 Row 44 Lost Advance Position... Check Ixxx.x French'
  433 = 'S2 433 Row 44 Lost Return Position... Check Ixxx.x Default' | German: 'S2 433 Row 44 Lost Return Position... Check Ixxx.x German' | French: 'S2 433 Row 44 Lost Return Position... Check Ixxx.x French'
  434 = 'S2 434 Row 44 Switch Fault... Check Ixxx.x / Ixxx.x Default' | German: 'S2 434 Row 44 Switch Fault... Check Ixxx.x / Ixxx.x German' | French: 'S2 434 Row 44 Switch Fault... Check Ixxx.x / Ixxx.x French'
  435 = 'S2 435 Row 44 Spare Message Default' | German: 'S2 435 Row 44 Spare Message German' | French: 'S2 435 Row 44 Spare Message French'
  436 = 'S2 436 Row 44 Spare Message Default' | German: 'S2 436 Row 44 Spare Message German' | French: 'S2 436 Row 44 Spare Message French'
  437 = 'S2 437 Row 44 Spare Message Default' | German: 'S2 437 Row 44 Spare Message German' | French: 'S2 437 Row 44 Spare Message French'
  438 = 'S2 438 Row 44 Spare Message Default' | German: 'S2 438 Row 44 Spare Message German' | French: 'S2 438 Row 44 Spare Message French'
  439 = 'S2 439 Row 44 Spare Message Default' | German: 'S2 439 Row 44 Spare Message German' | French: 'S2 439 Row 44 Spare Message French'
  440 = 'S2 440 Row 45 Failed To Advance.. Check Qxxx.x Default' | German: 'S2 440 Row 45 Failed To Advance.. Check Qxxx.x German' | French: 'S2 440 Row 45 Failed To Advance.. Check Qxxx.x French'
  441 = 'S2 441 Row 45 Failed To Return.. Check Qxxx.x Default' | German: 'S2 441 Row 45 Failed To Return.. Check Qxxx.x German' | French: 'S2 441 Row 45 Failed To Return.. Check Qxxx.x French'
  442 = 'S2 442 Row 45 Lost Advance Position... Check Ixxx.x Default' | German: 'S2 442 Row 45 Lost Advance Position... Check Ixxx.x German' | French: 'S2 442 Row 45 Lost Advance Position... Check Ixxx.x French'
  443 = 'S2 443 Row 45 Lost Return Position... Check Ixxx.x Default' | German: 'S2 443 Row 45 Lost Return Position... Check Ixxx.x German' | French: 'S2 443 Row 45 Lost Return Position... Check Ixxx.x French'
  444 = 'S2 444 Row 45 Switch Fault... Check Ixxx.x / Ixxx.x Default' | German: 'S2 444 Row 45 Switch Fault... Check Ixxx.x / Ixxx.x German' | French: 'S2 444 Row 45 Switch Fault... Check Ixxx.x / Ixxx.x French'
  445 = 'S2 445 Row 45 Spare Message Default' | German: 'S2 445 Row 45 Spare Message German' | French: 'S2 445 Row 45 Spare Message French'
  446 = 'S2 446 Row 45 Spare Message Default' | German: 'S2 446 Row 45 Spare Message German' | French: 'S2 446 Row 45 Spare Message French'
  447 = 'S2 447 Row 45 Spare Message Default' | German: 'S2 447 Row 45 Spare Message German' | French: 'S2 447 Row 45 Spare Message French'
  448 = 'S2 448 Row 45 Spare Message Default' | German: 'S2 448 Row 45 Spare Message German' | French: 'S2 448 Row 45 Spare Message French'
  449 = 'S2 449 Row 45 Spare Message Default' | German: 'S2 449 Row 45 Spare Message German' | French: 'S2 449 Row 45 Spare Message French'
  450 = 'S2 450 Row 46 Failed To Advance.. Check Qxxx.x Default' | German: 'S2 450 Row 46 Failed To Advance.. Check Qxxx.x German' | French: 'S2 450 Row 46 Failed To Advance.. Check Qxxx.x French'
  451 = 'S2 451 Row 46 Failed To Return.. Check Qxxx.x Default' | German: 'S2 451 Row 46 Failed To Return.. Check Qxxx.x German' | French: 'S2 451 Row 46 Failed To Return.. Check Qxxx.x French'
  452 = 'S2 452 Row 46 Lost Advance Position... Check Ixxx.x Default' | German: 'S2 452 Row 46 Lost Advance Position... Check Ixxx.x German' | French: 'S2 452 Row 46 Lost Advance Position... Check Ixxx.x French'
  453 = 'S2 453 Row 46 Lost Return Position... Check Ixxx.x Default' | German: 'S2 453 Row 46 Lost Return Position... Check Ixxx.x German' | French: 'S2 453 Row 46 Lost Return Position... Check Ixxx.x French'
  454 = 'S2 454 Row 46 Switch Fault... Check Ixxx.x / Ixxx.x Default' | German: 'S2 454 Row 46 Switch Fault... Check Ixxx.x / Ixxx.x German' | French: 'S2 454 Row 46 Switch Fault... Check Ixxx.x / Ixxx.x French'
  455 = 'S2 455 Row 46 Spare Message Default' | German: 'S2 455 Row 46 Spare Message German' | French: 'S2 455 Row 46 Spare Message French'
  456 = 'S2 456 Row 46 Spare Message Default' | German: 'S2 456 Row 46 Spare Message German' | French: 'S2 456 Row 46 Spare Message French'
  457 = 'S2 457 Row 46 Spare Message Default' | German: 'S2 457 Row 46 Spare Message German' | French: 'S2 457 Row 46 Spare Message French'
  458 = 'S2 458 Row 46 Spare Message Default' | German: 'S2 458 Row 46 Spare Message German' | French: 'S2 458 Row 46 Spare Message French'
  459 = 'S2 459 Row 46 Spare Message Default' | German: 'S2 459 Row 46 Spare Message German' | French: 'S2 459 Row 46 Spare Message French'
  460 = 'S2 460 Row 47 Failed To Advance.. Check Qxxx.x Default' | German: 'S2 460 Row 47 Failed To Advance.. Check Qxxx.x German' | French: 'S2 460 Row 47 Failed To Advance.. Check Qxxx.x French'
  461 = 'S2 461 Row 47 Failed To Return.. Check Qxxx.x Default' | German: 'S2 461 Row 47 Failed To Return.. Check Qxxx.x German' | French: 'S2 461 Row 47 Failed To Return.. Check Qxxx.x French'
  462 = 'S2 462 Row 47 Lost Advance Position... Check Ixxx.x Default' | German: 'S2 462 Row 47 Lost Advance Position... Check Ixxx.x German' | French: 'S2 462 Row 47 Lost Advance Position... Check Ixxx.x French'
  463 = 'S2 463 Row 47 Lost Return Position... Check Ixxx.x Default' | German: 'S2 463 Row 47 Lost Return Position... Check Ixxx.x German' | French: 'S2 463 Row 47 Lost Return Position... Check Ixxx.x French'
  464 = 'S2 464 Row 47 Switch Fault... Check Ixxx.x / Ixxx.x Default' | German: 'S2 464 Row 47 Switch Fault... Check Ixxx.x / Ixxx.x German' | French: 'S2 464 Row 47 Switch Fault... Check Ixxx.x / Ixxx.x French'
  465 = 'S2 465 Row 47 Spare Message Default' | German: 'S2 465 Row 47 Spare Message German' | French: 'S2 465 Row 47 Spare Message French'
  466 = 'S2 466 Row 47 Spare Message Default' | German: 'S2 466 Row 47 Spare Message German' | French: 'S2 466 Row 47 Spare Message French'
  467 = 'S2 467 Row 47 Spare Message Default' | German: 'S2 467 Row 47 Spare Message German' | French: 'S2 467 Row 47 Spare Message French'
  468 = 'S2 468 Row 47 Spare Message Default' | German: 'S2 468 Row 47 Spare Message German' | French: 'S2 468 Row 47 Spare Message French'
  469 = 'S2 469 Row 47 Spare Message Default' | German: 'S2 469 Row 47 Spare Message German' | French: 'S2 469 Row 47 Spare Message French'
  470 = 'S2 470 Row 48 Failed To Advance.. Check Qxxx.x Default' | German: 'S2 470 Row 48 Failed To Advance.. Check Qxxx.x German' | French: 'S2 470 Row 48 Failed To Advance.. Check Qxxx.x French'
  471 = 'S2 471 Row 48 Failed To Return.. Check Qxxx.x Default' | German: 'S2 471 Row 48 Failed To Return.. Check Qxxx.x German' | French: 'S2 471 Row 48 Failed To Return.. Check Qxxx.x French'
  472 = 'S2 472 Row 48 Lost Advance Position... Check Ixxx.x Default' | German: 'S2 472 Row 48 Lost Advance Position... Check Ixxx.x German' | French: 'S2 472 Row 48 Lost Advance Position... Check Ixxx.x French'
  473 = 'S2 473 Row 48 Lost Return Position... Check Ixxx.x Default' | German: 'S2 473 Row 48 Lost Return Position... Check Ixxx.x German' | French: 'S2 473 Row 48 Lost Return Position... Check Ixxx.x French'
  474 = 'S2 474 Row 48 Switch Fault... Check Ixxx.x / Ixxx.x Default' | German: 'S2 474 Row 48 Switch Fault... Check Ixxx.x / Ixxx.x German' | French: 'S2 474 Row 48 Switch Fault... Check Ixxx.x / Ixxx.x French'
  475 = 'S2 475 Row 48 Spare Message Default' | German: 'S2 475 Row 48 Spare Message German' | French: 'S2 475 Row 48 Spare Message French'
  476 = 'S2 476 Row 48 Spare Message Default' | German: 'S2 476 Row 48 Spare Message German' | French: 'S2 476 Row 48 Spare Message French'
  477 = 'S2 477 Row 48 Spare Message Default' | German: 'S2 477 Row 48 Spare Message German' | French: 'S2 477 Row 48 Spare Message French'
  478 = 'S2 478 Row 48 Spare Message Default' | German: 'S2 478 Row 48 Spare Message German' | French: 'S2 478 Row 48 Spare Message French'
  479 = 'S2 479 Row 48 Spare Message Default' | German: 'S2 479 Row 48 Spare Message German' | French: 'S2 479 Row 48 Spare Message French'
  480 = 'S2 480 Row 49 Failed To Advance.. Check Qxxx.x Default' | German: 'S2 480 Row 49 Failed To Advance.. Check Qxxx.x German' | French: 'S2 480 Row 49 Failed To Advance.. Check Qxxx.x French'
  481 = 'S2 481 Row 49 Failed To Return.. Check Qxxx.x Default' | German: 'S2 481 Row 49 Failed To Return.. Check Qxxx.x German' | French: 'S2 481 Row 49 Failed To Return.. Check Qxxx.x French'
  482 = 'S2 482 Row 49 Lost Advance Position... Check Ixxx.x Default' | German: 'S2 482 Row 49 Lost Advance Position... Check Ixxx.x German' | French: 'S2 482 Row 49 Lost Advance Position... Check Ixxx.x French'
  483 = 'S2 483 Row 49 Lost Return Position... Check Ixxx.x Default' | German: 'S2 483 Row 49 Lost Return Position... Check Ixxx.x German' | French: 'S2 483 Row 49 Lost Return Position... Check Ixxx.x French'
  484 = 'S2 484 Row 49 Switch Fault... Check Ixxx.x / Ixxx.x Default' | German: 'S2 484 Row 49 Switch Fault... Check Ixxx.x / Ixxx.x German' | French: 'S2 484 Row 49 Switch Fault... Check Ixxx.x / Ixxx.x French'
  485 = 'S2 485 Row 49 Spare Message Default' | German: 'S2 485 Row 49 Spare Message German' | French: 'S2 485 Row 49 Spare Message French'
  486 = 'S2 486 Row 49 Spare Message Default' | German: 'S2 486 Row 49 Spare Message German' | French: 'S2 486 Row 49 Spare Message French'
  487 = 'S2 487 Row 49 Spare Message Default' | German: 'S2 487 Row 49 Spare Message German' | French: 'S2 487 Row 49 Spare Message French'
  488 = 'S2 488 Row 49 Spare Message Default' | German: 'S2 488 Row 49 Spare Message German' | French: 'S2 488 Row 49 Spare Message French'
  489 = 'S2 489 Row 49 Spare Message Default' | German: 'S2 489 Row 49 Spare Message German' | French: 'S2 489 Row 49 Spare Message French'
  490 = 'S2 490 Row 50 Failed To Advance.. Check Qxxx.x Default' | German: 'S2 490 Row 50 Failed To Advance.. Check Qxxx.x German' | French: 'S2 490 Row 50 Failed To Advance.. Check Qxxx.x French'
  491 = 'S2 491 Row 50 Failed To Return.. Check Qxxx.x Default' | German: 'S2 491 Row 50 Failed To Return.. Check Qxxx.x German' | French: 'S2 491 Row 50 Failed To Return.. Check Qxxx.x French'
  492 = 'S2 492 Row 50 Lost Advance Position... Check Ixxx.x Default' | German: 'S2 492 Row 50 Lost Advance Position... Check Ixxx.x German' | French: 'S2 492 Row 50 Lost Advance Position... Check Ixxx.x French'
  493 = 'S2 493 Row 50 Lost Return Position... Check Ixxx.x Default' | German: 'S2 493 Row 50 Lost Return Position... Check Ixxx.x German' | French: 'S2 493 Row 50 Lost Return Position... Check Ixxx.x French'
  494 = 'S2 494 Row 50 Switch Fault... Check Ixxx.x / Ixxx.x Default' | German: 'S2 494 Row 50 Switch Fault... Check Ixxx.x / Ixxx.x German' | French: 'S2 494 Row 50 Switch Fault... Check Ixxx.x / Ixxx.x French'
  495 = 'S2 495 Row 50 Spare Message Default' | German: 'S2 495 Row 50 Spare Message German' | French: 'S2 495 Row 50 Spare Message French'
  496 = 'S2 496 Row 50 Spare Message Default' | German: 'S2 496 Row 50 Spare Message German' | French: 'S2 496 Row 50 Spare Message French'
  497 = 'S2 497 Row 50 Spare Message Default' | German: 'S2 497 Row 50 Spare Message German' | French: 'S2 497 Row 50 Spare Message French'
  498 = 'S2 498 Row 50 Spare Message Default' | German: 'S2 498 Row 50 Spare Message German' | French: 'S2 498 Row 50 Spare Message French'
  499 = 'S2 499 Row 50 Spare Message Default' | German: 'S2 499 Row 50 Spare Message German' | French: 'S2 499 Row 50 Spare Message French'
  500 = 'S2 500 Row 51 Failed To Advance.. Check Qxxx.x Default' | German: 'S2 500 Row 51 Failed To Advance.. Check Qxxx.x German' | French: 'S2 500 Row 51 Failed To Advance.. Check Qxxx.x French'
  501 = 'S2 501 Row 51 Failed To Return.. Check Qxxx.x Default' | German: 'S2 501 Row 51 Failed To Return.. Check Qxxx.x German' | French: 'S2 501 Row 51 Failed To Return.. Check Qxxx.x French'
  502 = 'S2 502 Row 51 Lost Advance Position... Check Ixxx.x Default' | German: 'S2 502 Row 51 Lost Advance Position... Check Ixxx.x German' | French: 'S2 502 Row 51 Lost Advance Position... Check Ixxx.x French'
  503 = 'S2 503 Row 51 Lost Return Position... Check Ixxx.x Default' | German: 'S2 503 Row 51 Lost Return Position... Check Ixxx.x German' | French: 'S2 503 Row 51 Lost Return Position... Check Ixxx.x French'
  504 = 'S2 504 Row 51 Switch Fault... Check Ixxx.x / Ixxx.x Default' | German: 'S2 504 Row 51 Switch Fault... Check Ixxx.x / Ixxx.x German' | French: 'S2 504 Row 51 Switch Fault... Check Ixxx.x / Ixxx.x French'
  505 = 'S2 505 Row 51 Spare Message Default' | German: 'S2 505 Row 51 Spare Message German' | French: 'S2 505 Row 51 Spare Message French'
  506 = 'S2 506 Row 51 Spare Message Default' | German: 'S2 506 Row 51 Spare Message German' | French: 'S2 506 Row 51 Spare Message French'
  507 = 'S2 507 Row 51 Spare Message Default' | German: 'S2 507 Row 51 Spare Message German' | French: 'S2 507 Row 51 Spare Message French'
  508 = 'S2 508 Row 51 Spare Message Default' | German: 'S2 508 Row 51 Spare Message German' | French: 'S2 508 Row 51 Spare Message French'
  509 = 'S2 509 Row 51 Spare Message Default' | German: 'S2 509 Row 51 Spare Message German' | French: 'S2 509 Row 51 Spare Message French'
  510 = 'S2 510 Row 52 Failed To Advance.. Check Qxxx.x Default' | German: 'S2 510 Row 52 Failed To Advance.. Check Qxxx.x German' | French: 'S2 510 Row 52 Failed To Advance.. Check Qxxx.x French'
  511 = 'S2 511 Row 52 Failed To Return.. Check Qxxx.x Default' | German: 'S2 511 Row 52 Failed To Return.. Check Qxxx.x German' | French: 'S2 511 Row 52 Failed To Return.. Check Qxxx.x French'
  512 = 'S2 512 Row 52 Lost Advance Position... Check Ixxx.x Default' | German: 'S2 512 Row 52 Lost Advance Position... Check Ixxx.x German' | French: 'S2 512 Row 52 Lost Advance Position... Check Ixxx.x French'
  513 = 'S2 513 Row 52 Lost Return Position... Check Ixxx.x Default' | German: 'S2 513 Row 52 Lost Return Position... Check Ixxx.x German' | French: 'S2 513 Row 52 Lost Return Position... Check Ixxx.x French'
  514 = 'S2 514 Row 52 Switch Fault... Check Ixxx.x / Ixxx.x Default' | German: 'S2 514 Row 52 Switch Fault... Check Ixxx.x / Ixxx.x German' | French: 'S2 514 Row 52 Switch Fault... Check Ixxx.x / Ixxx.x French'
  515 = 'S2 515 Row 52 Spare Message Default' | German: 'S2 515 Row 52 Spare Message German' | French: 'S2 515 Row 52 Spare Message French'
  516 = 'S2 516 Row 52 Spare Message Default' | German: 'S2 516 Row 52 Spare Message German' | French: 'S2 516 Row 52 Spare Message French'
  517 = 'S2 517 Row 52 Spare Message Default' | German: 'S2 517 Row 52 Spare Message German' | French: 'S2 517 Row 52 Spare Message French'
  518 = 'S2 518 Row 52 Spare Message Default' | German: 'S2 518 Row 52 Spare Message German' | French: 'S2 518 Row 52 Spare Message French'
  519 = 'S2 519 Row 52 Spare Message Default' | German: 'S2 519 Row 52 Spare Message German' | French: 'S2 519 Row 52 Spare Message French'
  520 = 'S2 520 Row 53 Failed To Advance.. Check Qxxx.x Default' | German: 'S2 520 Row 53 Failed To Advance.. Check Qxxx.x German' | French: 'S2 520 Row 53 Failed To Advance.. Check Qxxx.x French'
  521 = 'S2 521 Row 53 Failed To Return.. Check Qxxx.x Default' | German: 'S2 521 Row 53 Failed To Return.. Check Qxxx.x German' | French: 'S2 521 Row 53 Failed To Return.. Check Qxxx.x French'
  522 = 'S2 522 Row 53 Lost Advance Position... Check Ixxx.x Default' | German: 'S2 522 Row 53 Lost Advance Position... Check Ixxx.x German' | French: 'S2 522 Row 53 Lost Advance Position... Check Ixxx.x French'
  523 = 'S2 523 Row 53 Lost Return Position... Check Ixxx.x Default' | German: 'S2 523 Row 53 Lost Return Position... Check Ixxx.x German' | French: 'S2 523 Row 53 Lost Return Position... Check Ixxx.x French'
  524 = 'S2 524 Row 53 Switch Fault... Check Ixxx.x / Ixxx.x Default' | German: 'S2 524 Row 53 Switch Fault... Check Ixxx.x / Ixxx.x German' | French: 'S2 524 Row 53 Switch Fault... Check Ixxx.x / Ixxx.x French'
  525 = 'S2 525 Row 53 Spare Message Default' | German: 'S2 525 Row 53 Spare Message German' | French: 'S2 525 Row 53 Spare Message French'
  526 = 'S2 526 Row 53 Spare Message Default' | German: 'S2 526 Row 53 Spare Message German' | French: 'S2 526 Row 53 Spare Message French'
  527 = 'S2 527 Row 53 Spare Message Default' | German: 'S2 527 Row 53 Spare Message German' | French: 'S2 527 Row 53 Spare Message French'
  528 = 'S2 528 Row 53 Spare Message Default' | German: 'S2 528 Row 53 Spare Message German' | French: 'S2 528 Row 53 Spare Message French'
  529 = 'S2 529 Row 53 Spare Message Default' | German: 'S2 529 Row 53 Spare Message German' | French: 'S2 529 Row 53 Spare Message French'
  530 = 'S2 530 Row 54 Failed To Advance.. Check Qxxx.x Default' | German: 'S2 530 Row 54 Failed To Advance.. Check Qxxx.x German' | French: 'S2 530 Row 54 Failed To Advance.. Check Qxxx.x French'
  531 = 'S2 531 Row 54 Failed To Return.. Check Qxxx.x Default' | German: 'S2 531 Row 54 Failed To Return.. Check Qxxx.x German' | French: 'S2 531 Row 54 Failed To Return.. Check Qxxx.x French'
  532 = 'S2 532 Row 54 Lost Advance Position... Check Ixxx.x Default' | German: 'S2 532 Row 54 Lost Advance Position... Check Ixxx.x German' | French: 'S2 532 Row 54 Lost Advance Position... Check Ixxx.x French'
  533 = 'S2 533 Row 54 Lost Return Position... Check Ixxx.x Default' | German: 'S2 533 Row 54 Lost Return Position... Check Ixxx.x German' | French: 'S2 533 Row 54 Lost Return Position... Check Ixxx.x French'
  534 = 'S2 534 Row 54 Switch Fault... Check Ixxx.x / Ixxx.x Default' | German: 'S2 534 Row 54 Switch Fault... Check Ixxx.x / Ixxx.x German' | French: 'S2 534 Row 54 Switch Fault... Check Ixxx.x / Ixxx.x French'
  535 = 'S2 535 Row 54 Spare Message Default' | German: 'S2 535 Row 54 Spare Message German' | French: 'S2 535 Row 54 Spare Message French'
  536 = 'S2 536 Row 54 Spare Message Default' | German: 'S2 536 Row 54 Spare Message German' | French: 'S2 536 Row 54 Spare Message French'
  537 = 'S2 537 Row 54 Spare Message Default' | German: 'S2 537 Row 54 Spare Message German' | French: 'S2 537 Row 54 Spare Message French'
  538 = 'S2 538 Row 54 Spare Message Default' | German: 'S2 538 Row 54 Spare Message German' | French: 'S2 538 Row 54 Spare Message French'
  539 = 'S2 539 Row 54 Spare Message Default' | German: 'S2 539 Row 54 Spare Message German' | French: 'S2 539 Row 54 Spare Message French'
  540 = 'S2 540 Row 55 Failed To Advance.. Check Qxxx.x Default' | German: 'S2 540 Row 55 Failed To Advance.. Check Qxxx.x German' | French: 'S2 540 Row 55 Failed To Advance.. Check Qxxx.x French'
  541 = 'S2 541 Row 55 Failed To Return.. Check Qxxx.x Default' | German: 'S2 541 Row 55 Failed To Return.. Check Qxxx.x German' | French: 'S2 541 Row 55 Failed To Return.. Check Qxxx.x French'
  542 = 'S2 542 Row 55 Lost Advance Position... Check Ixxx.x Default' | German: 'S2 542 Row 55 Lost Advance Position... Check Ixxx.x German' | French: 'S2 542 Row 55 Lost Advance Position... Check Ixxx.x French'
  543 = 'S2 543 Row 55 Lost Return Position... Check Ixxx.x Default' | German: 'S2 543 Row 55 Lost Return Position... Check Ixxx.x German' | French: 'S2 543 Row 55 Lost Return Position... Check Ixxx.x French'
  544 = 'S2 544 Row 55 Switch Fault... Check Ixxx.x / Ixxx.x Default' | German: 'S2 544 Row 55 Switch Fault... Check Ixxx.x / Ixxx.x German' | French: 'S2 544 Row 55 Switch Fault... Check Ixxx.x / Ixxx.x French'
  545 = 'S2 545 Row 55 Spare Message Default' | German: 'S2 545 Row 55 Spare Message German' | French: 'S2 545 Row 55 Spare Message French'
  546 = 'S2 546 Row 55 Spare Message Default' | German: 'S2 546 Row 55 Spare Message German' | French: 'S2 546 Row 55 Spare Message French'
  547 = 'S2 547 Row 55 Spare Message Default' | German: 'S2 547 Row 55 Spare Message German' | French: 'S2 547 Row 55 Spare Message French'
  548 = 'S2 548 Row 55 Spare Message Default' | German: 'S2 548 Row 55 Spare Message German' | French: 'S2 548 Row 55 Spare Message French'
  549 = 'S2 549 Row 55 Spare Message Default' | German: 'S2 549 Row 55 Spare Message German' | French: 'S2 549 Row 55 Spare Message French'
  550 = 'S2 550 Row 56 Failed To Advance.. Check Qxxx.x Default' | German: 'S2 550 Row 56 Failed To Advance.. Check Qxxx.x German' | French: 'S2 550 Row 56 Failed To Advance.. Check Qxxx.x French'
  551 = 'S2 551 Row 56 Failed To Return.. Check Qxxx.x Default' | German: 'S2 551 Row 56 Failed To Return.. Check Qxxx.x German' | French: 'S2 551 Row 56 Failed To Return.. Check Qxxx.x French'
  552 = 'S2 552 Row 56 Lost Advance Position... Check Ixxx.x Default' | German: 'S2 552 Row 56 Lost Advance Position... Check Ixxx.x German' | French: 'S2 552 Row 56 Lost Advance Position... Check Ixxx.x French'
  553 = 'S2 553 Row 56 Lost Return Position... Check Ixxx.x Default' | German: 'S2 553 Row 56 Lost Return Position... Check Ixxx.x German' | French: 'S2 553 Row 56 Lost Return Position... Check Ixxx.x French'
  554 = 'S2 554 Row 56 Switch Fault... Check Ixxx.x / Ixxx.x Default' | German: 'S2 554 Row 56 Switch Fault... Check Ixxx.x / Ixxx.x German' | French: 'S2 554 Row 56 Switch Fault... Check Ixxx.x / Ixxx.x French'
  555 = 'S2 555 Row 56 Spare Message Default' | German: 'S2 555 Row 56 Spare Message German' | French: 'S2 555 Row 56 Spare Message French'
  556 = 'S2 556 Row 56 Spare Message Default' | German: 'S2 556 Row 56 Spare Message German' | French: 'S2 556 Row 56 Spare Message French'
  557 = 'S2 557 Row 56 Spare Message Default' | German: 'S2 557 Row 56 Spare Message German' | French: 'S2 557 Row 56 Spare Message French'
  558 = 'S2 558 Row 56 Spare Message Default' | German: 'S2 558 Row 56 Spare Message German' | French: 'S2 558 Row 56 Spare Message French'
  559 = 'S2 559 Row 56 Spare Message Default' | German: 'S2 559 Row 56 Spare Message German' | French: 'S2 559 Row 56 Spare Message French'
  560 = 'S2 560 Row 57 Failed To Advance.. Check Qxxx.x Default' | German: 'S2 560 Row 57 Failed To Advance.. Check Qxxx.x German' | French: 'S2 560 Row 57 Failed To Advance.. Check Qxxx.x French'
  561 = 'S2 561 Row 57 Failed To Return.. Check Qxxx.x Default' | German: 'S2 561 Row 57 Failed To Return.. Check Qxxx.x German' | French: 'S2 561 Row 57 Failed To Return.. Check Qxxx.x French'
  562 = 'S2 562 Row 57 Lost Advance Position... Check Ixxx.x Default' | German: 'S2 562 Row 57 Lost Advance Position... Check Ixxx.x German' | French: 'S2 562 Row 57 Lost Advance Position... Check Ixxx.x French'
  563 = 'S2 563 Row 57 Lost Return Position... Check Ixxx.x Default' | German: 'S2 563 Row 57 Lost Return Position... Check Ixxx.x German' | French: 'S2 563 Row 57 Lost Return Position... Check Ixxx.x French'
  564 = 'S2 564 Row 57 Switch Fault... Check Ixxx.x / Ixxx.x Default' | German: 'S2 564 Row 57 Switch Fault... Check Ixxx.x / Ixxx.x German' | French: 'S2 564 Row 57 Switch Fault... Check Ixxx.x / Ixxx.x French'
  565 = 'S2 565 Row 57 Spare Message Default' | German: 'S2 565 Row 57 Spare Message German' | French: 'S2 565 Row 57 Spare Message French'
  566 = 'S2 566 Row 57 Spare Message Default' | German: 'S2 566 Row 57 Spare Message German' | French: 'S2 566 Row 57 Spare Message French'
  567 = 'S2 567 Row 57 Spare Message Default' | German: 'S2 567 Row 57 Spare Message German' | French: 'S2 567 Row 57 Spare Message French'
  568 = 'S2 568 Row 57 Spare Message Default' | German: 'S2 568 Row 57 Spare Message German' | French: 'S2 568 Row 57 Spare Message French'
  569 = 'S2 569 Row 57 Spare Message Default' | German: 'S2 569 Row 57 Spare Message German' | French: 'S2 569 Row 57 Spare Message French'
  570 = 'S2 570 Row 58 Failed To Advance.. Check Qxxx.x Default' | German: 'S2 570 Row 58 Failed To Advance.. Check Qxxx.x German' | French: 'S2 570 Row 58 Failed To Advance.. Check Qxxx.x French'
  571 = 'S2 571 Row 58 Failed To Return.. Check Qxxx.x Default' | German: 'S2 571 Row 58 Failed To Return.. Check Qxxx.x German' | French: 'S2 571 Row 58 Failed To Return.. Check Qxxx.x French'
  572 = 'S2 572 Row 58 Lost Advance Position... Check Ixxx.x Default' | German: 'S2 572 Row 58 Lost Advance Position... Check Ixxx.x German' | French: 'S2 572 Row 58 Lost Advance Position... Check Ixxx.x French'
  573 = 'S2 573 Row 58 Lost Return Position... Check Ixxx.x Default' | German: 'S2 573 Row 58 Lost Return Position... Check Ixxx.x German' | French: 'S2 573 Row 58 Lost Return Position... Check Ixxx.x French'
  574 = 'S2 574 Row 58 Switch Fault... Check Ixxx.x / Ixxx.x Default' | German: 'S2 574 Row 58 Switch Fault... Check Ixxx.x / Ixxx.x German' | French: 'S2 574 Row 58 Switch Fault... Check Ixxx.x / Ixxx.x French'
  575 = 'S2 575 Row 58 Spare Message Default' | German: 'S2 575 Row 58 Spare Message German' | French: 'S2 575 Row 58 Spare Message French'
  576 = 'S2 576 Row 58 Spare Message Default' | German: 'S2 576 Row 58 Spare Message German' | French: 'S2 576 Row 58 Spare Message French'
  577 = 'S2 577 Row 58 Spare Message Default' | German: 'S2 577 Row 58 Spare Message German' | French: 'S2 577 Row 58 Spare Message French'
  578 = 'S2 578 Row 58 Spare Message Default' | German: 'S2 578 Row 58 Spare Message German' | French: 'S2 578 Row 58 Spare Message French'
  579 = 'S2 579 Row 58 Spare Message Default' | German: 'S2 579 Row 58 Spare Message German' | French: 'S2 579 Row 58 Spare Message French'
  580 = 'S2 580 Row 59 Failed To Advance.. Check Qxxx.x Default' | German: 'S2 580 Row 59 Failed To Advance.. Check Qxxx.x German' | French: 'S2 580 Row 59 Failed To Advance.. Check Qxxx.x French'
  581 = 'S2 581 Row 59 Failed To Return.. Check Qxxx.x Default' | German: 'S2 581 Row 59 Failed To Return.. Check Qxxx.x German' | French: 'S2 581 Row 59 Failed To Return.. Check Qxxx.x French'
  582 = 'S2 582 Row 59 Lost Advance Position... Check Ixxx.x Default' | German: 'S2 582 Row 59 Lost Advance Position... Check Ixxx.x German' | French: 'S2 582 Row 59 Lost Advance Position... Check Ixxx.x French'
